REGION Network 20: Check connect giữa PLC với Server và HMI
   RUNG wire#powerrail
      Contact( "AlwaysTRUE" )
      "CheckConnectPLCServer_DB"(Signal := wire#w1, "Timeout(s)" := 60, Status => "DB_DataHMI".StatusConnectServer)
   END_RUNG
   RUNG wire#powerrail
      Contact( "AlwaysTRUE" )
      Contact( "DB_Server".ConnectPLC )
   END_RUNG wire#w1
   RUNG wire#powerrail
      Contact( "AlwaysTRUE" )
      Contact( "DB_Server".ConnectPLC )
      R_Coil( "DB_Server".ConnectPLC )
   END_RUNG
   RUNG wire#powerrail
      Contact( "AlwaysTRUE" )
      wire#w2
      "CreatePulse_DB_CheckConnectHMI"("pulse_on(x1ms)" := 1000, "pulse_off(x1ms)" := 1000, pulse => #pulse_check_connect_hmi)
   END_RUNG
   RUNG wire#w2
      P_Contact(operand := #pulse_check_connect_hmi, bit := "PulseP_Check_ConnectHmi")
      S_Coil( "DB_DataHMI".StatusConnectController )
   END_RUNG
   // the same network as SCL:
   IF "AlwaysTRUE" THEN
       "CheckConnectPLCServer_DB"(Signal := "AlwaysTRUE" AND "DB_Server".ConnectPLC,   // "CheckConnectPLCServer"
                               "Timeout(s)" := 60,
                               Status => "DB_DataHMI".StatusConnectServer);
   END_IF;
   IF "AlwaysTRUE" AND "DB_Server".ConnectPLC THEN "DB_Server".ConnectPLC := FALSE; END_IF;
   #_w1 := "AlwaysTRUE";
   IF #_w1 THEN
       "CreatePulse_DB_CheckConnectHMI"("pulse_on(x1ms)" := 1000,   // "CreatePulse"
                               "pulse_off(x1ms)" := 1000,
                               pulse => #pulse_check_connect_hmi);
   END_IF;
   #_w2 := #_w1 AND #pulse_check_connect_hmi AND NOT "PulseP_Check_ConnectHmi";   // rising edge of #pulse_check_connect_hmi
   "PulseP_Check_ConnectHmi" := #pulse_check_connect_hmi;
   IF #_w2 THEN "DB_DataHMI".StatusConnectController := TRUE; END_IF;
END_REGION

REGION Network 21: Reset Counter khi qua ca
   RUNG wire#powerrail
      Contact( "AlwaysTRUE" )
      Contact( "DB_Server".EventResetCounterInShift )
      wire#w1
      Add(in1 := "TagTest".NumberServerResetCounter, in2 := 1, out => "TagTest".NumberServerResetCounter)
      Move(in := 0, out1 => "DB_Machine".CounterMachineInShift)
      "ClearBufferLossInShift"()
   END_RUNG
   RUNG wire#w1
      R_Coil( "DB_Server".EventResetCounterInShift )
   END_RUNG
   // the same network as SCL:
   IF "AlwaysTRUE" AND "DB_Server".EventResetCounterInShift THEN
       "TagTest".NumberServerResetCounter := "TagTest".NumberServerResetCounter + 1;
       "DB_Machine".CounterMachineInShift := 0;
   END_IF;
   #_w1 := "AlwaysTRUE" AND "DB_Server".EventResetCounterInShift;
   IF #_w1 THEN
       "ClearBufferLossInShift"();
       "DB_Server".EventResetCounterInShift := FALSE;
   END_IF;
END_REGION

REGION Network 22: //////////////////End//////////////////
END_REGION

REGION Network 23: Test tính Speed
END_REGION

REGION Network 24 (SCL): Random Buffer Test
   IF "TagTest".TestRandomSparePart THEN
       "DB_Server".PageDataSparePart.MaxPage := 10;
       "DB_Server".ActionSearchLossSparePart := 2;
       "DB_Server".PageDataSparePart.TotalData := "DB_Server".PageDataSparePart.MaxPage * 30;

       FOR #index_for := 1 TO 30 DO
           #id_test := ("DB_Server".PageDataSparePart.PageCurrent - 1) * 30 + #index_for;

           "BufferServerSend".buffer_spare_part[#index_for].name := CONCAT(IN1 := 'Thiet bi: ', IN2 := UDINT_TO_STRING(#id_test));
           "BufferServerSend".buffer_spare_part[#index_for].start_time := "GlobalDB_RTC".RTC_Local;
           "BufferServerSend".buffer_spare_part[#index_for].end_time := "GlobalDB_RTC".RTC_Local;
           "BufferServerSend".buffer_spare_part[#index_for].product_count := #id_test;
       END_FOR;
   END_IF;


   IF "TagTest".TestRandomHistorical THEN
       FOR #index_for := 1 TO 50 DO
           #id_test := ("DB_Server".PageHistorical.PageCurrent - 1) * 50 + #index_for;

           "BuffersLoss_DB".buffer_loss_in_historical[#index_for].id := #id_test;
           "BuffersLoss_DB".buffer_loss_in_historical[#index_for].duration := #id_test * 10;
           "BuffersLoss_DB".buffer_loss_in_historical[#index_for].startTime := "GlobalDB_RTC".RTC_Local;
           "BuffersLoss_DB".buffer_loss_in_historical[#index_for].endTime := "GlobalDB_RTC".RTC_Local;
           "BuffersLoss_DB".buffer_loss_in_historical[#index_for].losscode := 0;
           "BuffersLoss_DB".buffer_loss_in_historical[#index_for].statusServer := 0;
       END_FOR;
   END_IF;
END_REGION

REGION Network 25: Clear Buffer To Test
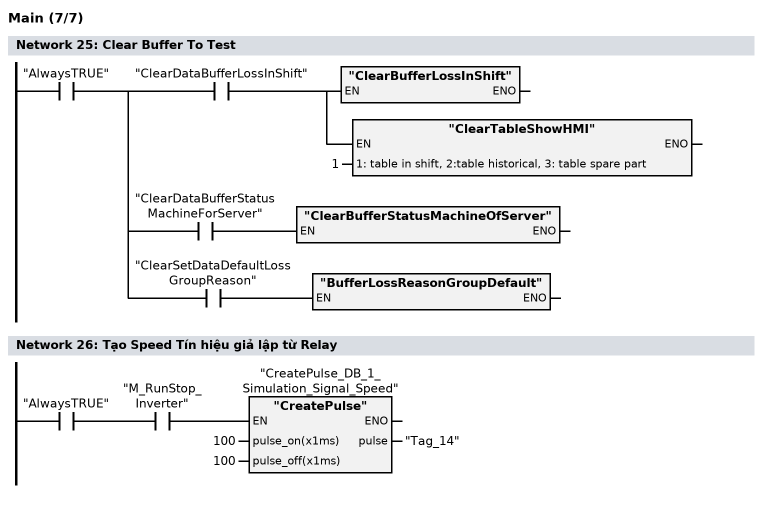
   RUNG wire#powerrail
      Contact( "AlwaysTRUE" )
      wire#w1
      Contact( "ClearDataBufferLossInShift" )
      wire#w2
      "ClearBufferLossInShift"()
   END_RUNG
   RUNG wire#w2
      "ClearTableShowHMI"("1: table in shift, 2:table historical, 3: table spare part" := 1)
   END_RUNG
   RUNG wire#w1
      Contact( "ClearDataBufferStatusMachineForServer" )
      "ClearBufferStatusMachineOfServer"()
   END_RUNG
   RUNG wire#w1
      Contact( "ClearSetDataDefaultLossGroupReason" )
      "BufferLossReasonGroupDefault"()
   END_RUNG
   // the same network as SCL:
   #_w1 := "AlwaysTRUE";
   #_w2 := "AlwaysTRUE" AND "ClearDataBufferLossInShift";
   IF #_w2 THEN
       "ClearBufferLossInShift"();
       "ClearTableShowHMI"("1: table in shift, 2:table historical, 3: table spare part" := 1);
   END_IF;
   IF #_w1 AND "ClearDataBufferStatusMachineForServer" THEN "ClearBufferStatusMachineOfServer"(); END_IF;
   IF #_w1 AND "ClearSetDataDefaultLossGroupReason" THEN "BufferLossReasonGroupDefault"(); END_IF;
END_REGION

REGION Network 26: Tạo Speed Tín hiệu giả lập từ Relay
   RUNG wire#powerrail
      Contact( "AlwaysTRUE" )
      Contact( "M_RunStop_Inverter" )
      "CreatePulse_DB_1_Simulation_Signal_Speed"("pulse_on(x1ms)" := 100, "pulse_off(x1ms)" := 100, pulse => "Tag_14")
   END_RUNG
   // the same network as SCL:
   IF "AlwaysTRUE" AND "M_RunStop_Inverter" THEN
       "CreatePulse_DB_1_Simulation_Signal_Speed"("pulse_on(x1ms)" := 100,   // "CreatePulse"
                               "pulse_off(x1ms)" := 100,
                               pulse => "Tag_14");
   END_IF;
END_REGION
END_ORGANIZATION_BLOCK

ORGANIZATION_BLOCK "InterrupTimer10ms(Simulation)"   // OB30, LAD, CyclicInterrupt
{ S7_Optimized_Access := 'TRUE' }
VERSION : 0.1
   VAR_INPUT
      Initial_Call : Bool;   // Initial call of this OB
      Event_Count : Int;   // Events discarded
   END_VAR
BEGIN

REGION Network 1: Tạo xung simulation cho sensors
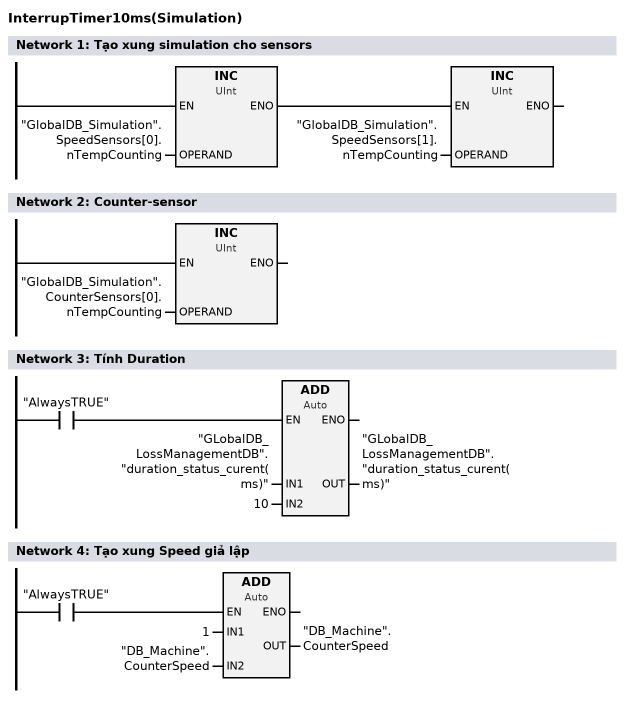
   RUNG wire#powerrail
      { S7_Templates := "DestType := UInt" } Inc( "GlobalDB_Simulation".SpeedSensors[0].nTempCounting )
      { S7_Templates := "DestType := UInt" } Inc( "GlobalDB_Simulation".SpeedSensors[1].nTempCounting )
   END_RUNG
   // the same network as SCL:
   "GlobalDB_Simulation".SpeedSensors[0].nTempCounting := "GlobalDB_Simulation".SpeedSensors[0].nTempCounting + 1;
   "GlobalDB_Simulation".SpeedSensors[1].nTempCounting := "GlobalDB_Simulation".SpeedSensors[1].nTempCounting + 1;
END_REGION

REGION Network 2: Counter-sensor
   RUNG wire#powerrail
      { S7_Templates := "DestType := UInt" } Inc( "GlobalDB_Simulation".CounterSensors[0].nTempCounting )
   END_RUNG
   // the same network as SCL:
   "GlobalDB_Simulation".CounterSensors[0].nTempCounting := "GlobalDB_Simulation".CounterSensors[0].nTempCounting + 1;
END_REGION

REGION Network 3: Tính Duration
   RUNG wire#powerrail
      Contact( "AlwaysTRUE" )
      Add(in1 := "GLobalDB_LossManagementDB"."duration_status_curent(ms)", in2 := 10, out => "GLobalDB_LossManagementDB"."duration_status_curent(ms)")
   END_RUNG
   // the same network as SCL:
   IF "AlwaysTRUE" THEN
       "GLobalDB_LossManagementDB"."duration_status_curent(ms)" := "GLobalDB_LossManagementDB"."duration_status_curent(ms)" + 10;
   END_IF;
END_REGION

REGION Network 4: Tạo xung Speed giả lập
   RUNG wire#powerrail
      Contact( "AlwaysTRUE" )
      Add(in1 := 1, in2 := "DB_Machine".CounterSpeed, out => "DB_Machine".CounterSpeed)
   END_RUNG
   // the same network as SCL:
   IF "AlwaysTRUE" THEN "DB_Machine".CounterSpeed := 1 + "DB_Machine".CounterSpeed; END_IF;
END_REGION
END_ORGANIZATION_BLOCK

ORGANIZATION_BLOCK "Interrupt Analog Cyclic"   // OB31, LAD, CyclicInterrupt
{ S7_Optimized_Access := 'TRUE' }
VERSION : 0.1
   VAR_INPUT
      Initial_Call : Bool;   // Initial call of this OB
      Event_Count : Int;   // Events discarded
   END_VAR
   VAR CONSTANT
      MAX_IDX : Int := 3;
   END_VAR
   VAR_TEMP   // added for the SCL form of the ladder/FBD networks
      _w1 : Bool;
      _w2 : Bool;
   END_VAR
BEGIN

REGION Network 1: Check Index
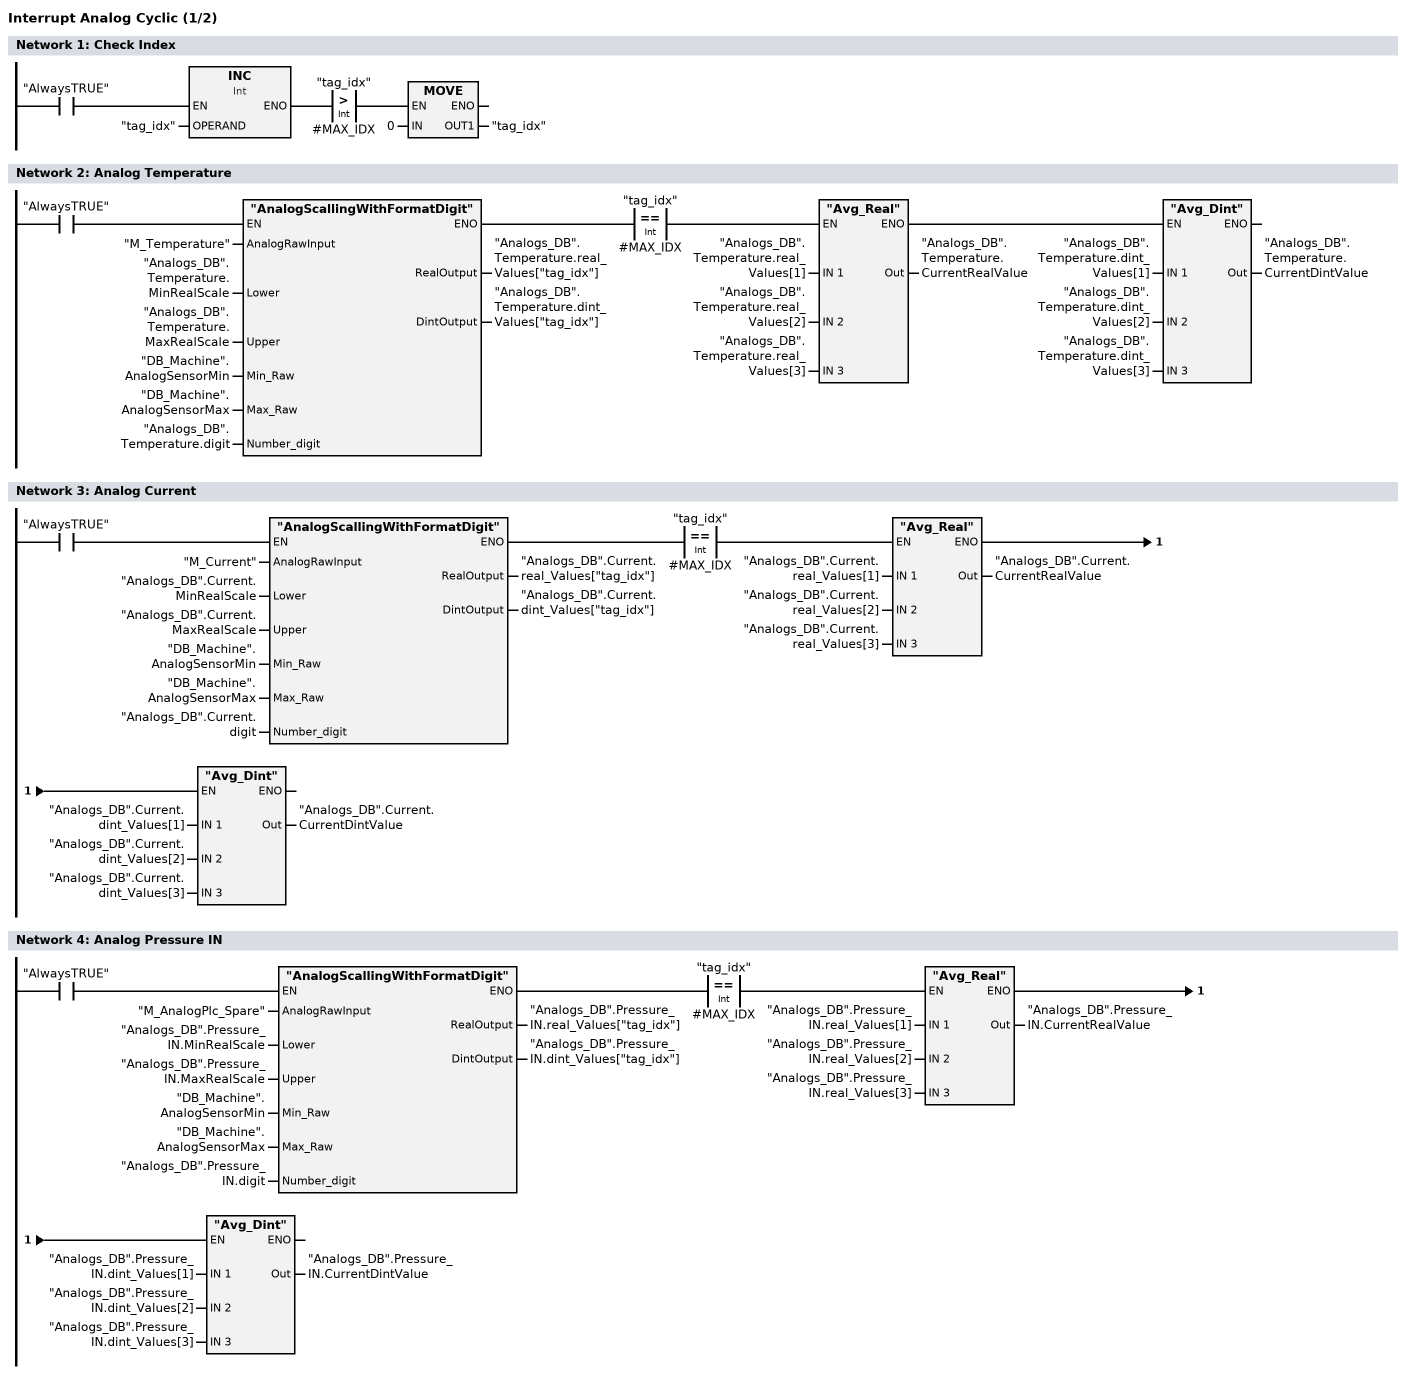
   RUNG wire#powerrail
      Contact( "AlwaysTRUE" )
      { S7_Templates := "DestType := Int" } Inc( "tag_idx" )
      { S7_Templates := "SrcType := Int" } GT_Contact(in1 := "tag_idx", in2 := #MAX_IDX)
      Move(in := 0, out1 => "tag_idx")
   END_RUNG
   // the same network as SCL:
   IF "AlwaysTRUE" THEN "tag_idx" := "tag_idx" + 1; END_IF;
   IF "AlwaysTRUE" AND ("tag_idx" > #MAX_IDX) THEN "tag_idx" := 0; END_IF;
END_REGION

REGION Network 2: Analog Temperature
   RUNG wire#powerrail
      Contact( "AlwaysTRUE" )
      "AnalogScallingWithFormatDigit"(AnalogRawInput := "M_Temperature", Lower := "Analogs_DB".Temperature.MinRealScale, Upper := "Analogs_DB".Temperature.MaxRealScale, Min_Raw := "DB_Machine".AnalogSensorMin, Max_Raw := "DB_Machine".AnalogSensorMax, Number_digit := "Analogs_DB".Temperature.digit, RealOutput => "Analogs_DB".Temperature.real_Values["tag_idx"], DintOutput => "Analogs_DB".Temperature.dint_Values["tag_idx"])
      { S7_Templates := "SrcType := Int" } EQ_Contact(in1 := "tag_idx", in2 := #MAX_IDX)
      "Avg_Real"("IN 1" := "Analogs_DB".Temperature.real_Values[1], "IN 2" := "Analogs_DB".Temperature.real_Values[2], "IN 3" := "Analogs_DB".Temperature.real_Values[3], Out => "Analogs_DB".Temperature.CurrentRealValue)
      "Avg_Dint"("IN 1" := "Analogs_DB".Temperature.dint_Values[1], "IN 2" := "Analogs_DB".Temperature.dint_Values[2], "IN 3" := "Analogs_DB".Temperature.dint_Values[3], Out => "Analogs_DB".Temperature.CurrentDintValue)
   END_RUNG
   // the same network as SCL:
   "AnalogScallingWithFormatDigit"(EN := "AlwaysTRUE",
                           AnalogRawInput := "M_Temperature",
                           Lower := "Analogs_DB".Temperature.MinRealScale,
                           Upper := "Analogs_DB".Temperature.MaxRealScale,
                           Min_Raw := "DB_Machine".AnalogSensorMin,
                           Max_Raw := "DB_Machine".AnalogSensorMax,
                           Number_digit := "Analogs_DB".Temperature.digit,
                           RealOutput => "Analogs_DB".Temperature.real_Values["tag_idx"],
                           DintOutput => "Analogs_DB".Temperature.dint_Values["tag_idx"],
                           ENO => #_w1);
   "Avg_Real"(EN := #_w1 AND ("tag_idx" = #MAX_IDX),
              "IN 1" := "Analogs_DB".Temperature.real_Values[1],
              "IN 2" := "Analogs_DB".Temperature.real_Values[2],
              "IN 3" := "Analogs_DB".Temperature.real_Values[3],
              Out => "Analogs_DB".Temperature.CurrentRealValue,
              ENO => #_w2);
   IF #_w2 THEN
       "Avg_Dint"("IN 1" := "Analogs_DB".Temperature.dint_Values[1],
                  "IN 2" := "Analogs_DB".Temperature.dint_Values[2],
                  "IN 3" := "Analogs_DB".Temperature.dint_Values[3],
                  Out => "Analogs_DB".Temperature.CurrentDintValue);
   END_IF;
END_REGION

REGION Network 3: Analog Current
   RUNG wire#powerrail
      Contact( "AlwaysTRUE" )
      "AnalogScallingWithFormatDigit"(AnalogRawInput := "M_Current", Lower := "Analogs_DB".Current.MinRealScale, Upper := "Analogs_DB".Current.MaxRealScale, Min_Raw := "DB_Machine".AnalogSensorMin, Max_Raw := "DB_Machine".AnalogSensorMax, Number_digit := "Analogs_DB".Current.digit, RealOutput => "Analogs_DB".Current.real_Values["tag_idx"], DintOutput => "Analogs_DB".Current.dint_Values["tag_idx"])
      { S7_Templates := "SrcType := Int" } EQ_Contact(in1 := "tag_idx", in2 := #MAX_IDX)
      "Avg_Real"("IN 1" := "Analogs_DB".Current.real_Values[1], "IN 2" := "Analogs_DB".Current.real_Values[2], "IN 3" := "Analogs_DB".Current.real_Values[3], Out => "Analogs_DB".Current.CurrentRealValue)
      "Avg_Dint"("IN 1" := "Analogs_DB".Current.dint_Values[1], "IN 2" := "Analogs_DB".Current.dint_Values[2], "IN 3" := "Analogs_DB".Current.dint_Values[3], Out => "Analogs_DB".Current.CurrentDintValue)
   END_RUNG
   // the same network as SCL:
   "AnalogScallingWithFormatDigit"(EN := "AlwaysTRUE",
                           AnalogRawInput := "M_Current",
                           Lower := "Analogs_DB".Current.MinRealScale,
                           Upper := "Analogs_DB".Current.MaxRealScale,
                           Min_Raw := "DB_Machine".AnalogSensorMin,
                           Max_Raw := "DB_Machine".AnalogSensorMax,
                           Number_digit := "Analogs_DB".Current.digit,
                           RealOutput => "Analogs_DB".Current.real_Values["tag_idx"],
                           DintOutput => "Analogs_DB".Current.dint_Values["tag_idx"],
                           ENO => #_w1);
   "Avg_Real"(EN := #_w1 AND ("tag_idx" = #MAX_IDX),
              "IN 1" := "Analogs_DB".Current.real_Values[1],
              "IN 2" := "Analogs_DB".Current.real_Values[2],
              "IN 3" := "Analogs_DB".Current.real_Values[3],
              Out => "Analogs_DB".Current.CurrentRealValue,
              ENO => #_w2);
   IF #_w2 THEN
       "Avg_Dint"("IN 1" := "Analogs_DB".Current.dint_Values[1],
                  "IN 2" := "Analogs_DB".Current.dint_Values[2],
                  "IN 3" := "Analogs_DB".Current.dint_Values[3],
                  Out => "Analogs_DB".Current.CurrentDintValue);
   END_IF;
END_REGION

REGION Network 4: Analog Pressure IN
   RUNG wire#powerrail
      Contact( "AlwaysTRUE" )
      "AnalogScallingWithFormatDigit"(AnalogRawInput := "M_AnalogPlc_Spare", Lower := "Analogs_DB".Pressure_IN.MinRealScale, Upper := "Analogs_DB".Pressure_IN.MaxRealScale, Min_Raw := "DB_Machine".AnalogSensorMin, Max_Raw := "DB_Machine".AnalogSensorMax, Number_digit := "Analogs_DB".Pressure_IN.digit, RealOutput => "Analogs_DB".Pressure_IN.real_Values["tag_idx"], DintOutput => "Analogs_DB".Pressure_IN.dint_Values["tag_idx"])
      { S7_Templates := "SrcType := Int" } EQ_Contact(in1 := "tag_idx", in2 := #MAX_IDX)
      "Avg_Real"("IN 1" := "Analogs_DB".Pressure_IN.real_Values[1], "IN 2" := "Analogs_DB".Pressure_IN.real_Values[2], "IN 3" := "Analogs_DB".Pressure_IN.real_Values[3], Out => "Analogs_DB".Pressure_IN.CurrentRealValue)
      "Avg_Dint"("IN 1" := "Analogs_DB".Pressure_IN.dint_Values[1], "IN 2" := "Analogs_DB".Pressure_IN.dint_Values[2], "IN 3" := "Analogs_DB".Pressure_IN.dint_Values[3], Out => "Analogs_DB".Pressure_IN.CurrentDintValue)
   END_RUNG
   // the same network as SCL:
   "AnalogScallingWithFormatDigit"(EN := "AlwaysTRUE",
                           AnalogRawInput := "M_AnalogPlc_Spare",
                           Lower := "Analogs_DB".Pressure_IN.MinRealScale,
                           Upper := "Analogs_DB".Pressure_IN.MaxRealScale,
                           Min_Raw := "DB_Machine".AnalogSensorMin,
                           Max_Raw := "DB_Machine".AnalogSensorMax,
                           Number_digit := "Analogs_DB".Pressure_IN.digit,
                           RealOutput => "Analogs_DB".Pressure_IN.real_Values["tag_idx"],
                           DintOutput => "Analogs_DB".Pressure_IN.dint_Values["tag_idx"],
                           ENO => #_w1);
   "Avg_Real"(EN := #_w1 AND ("tag_idx" = #MAX_IDX),
              "IN 1" := "Analogs_DB".Pressure_IN.real_Values[1],
              "IN 2" := "Analogs_DB".Pressure_IN.real_Values[2],
              "IN 3" := "Analogs_DB".Pressure_IN.real_Values[3],
              Out => "Analogs_DB".Pressure_IN.CurrentRealValue,
              ENO => #_w2);
   IF #_w2 THEN
       "Avg_Dint"("IN 1" := "Analogs_DB".Pressure_IN.dint_Values[1],
                  "IN 2" := "Analogs_DB".Pressure_IN.dint_Values[2],
                  "IN 3" := "Analogs_DB".Pressure_IN.dint_Values[3],
                  Out => "Analogs_DB".Pressure_IN.CurrentDintValue);
   END_IF;
END_REGION

REGION Network 5: Analog Pressure OUT
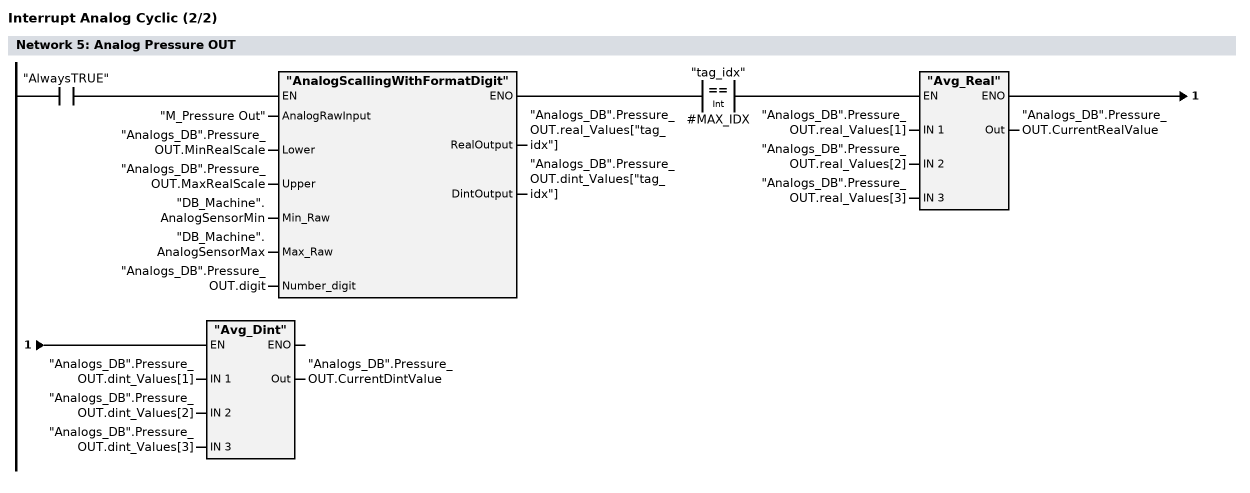
   RUNG wire#powerrail
      Contact( "AlwaysTRUE" )
      "AnalogScallingWithFormatDigit"(AnalogRawInput := "M_Pressure Out", Lower := "Analogs_DB".Pressure_OUT.MinRealScale, Upper := "Analogs_DB".Pressure_OUT.MaxRealScale, Min_Raw := "DB_Machine".AnalogSensorMin, Max_Raw := "DB_Machine".AnalogSensorMax, Number_digit := "Analogs_DB".Pressure_OUT.digit, RealOutput => "Analogs_DB".Pressure_OUT.real_Values["tag_idx"], DintOutput => "Analogs_DB".Pressure_OUT.dint_Values["tag_idx"])
      { S7_Templates := "SrcType := Int" } EQ_Contact(in1 := "tag_idx", in2 := #MAX_IDX)
      "Avg_Real"("IN 1" := "Analogs_DB".Pressure_OUT.real_Values[1], "IN 2" := "Analogs_DB".Pressure_OUT.real_Values[2], "IN 3" := "Analogs_DB".Pressure_OUT.real_Values[3], Out => "Analogs_DB".Pressure_OUT.CurrentRealValue)
      "Avg_Dint"("IN 1" := "Analogs_DB".Pressure_OUT.dint_Values[1], "IN 2" := "Analogs_DB".Pressure_OUT.dint_Values[2], "IN 3" := "Analogs_DB".Pressure_OUT.dint_Values[3], Out => "Analogs_DB".Pressure_OUT.CurrentDintValue)
   END_RUNG
   // the same network as SCL:
   "AnalogScallingWithFormatDigit"(EN := "AlwaysTRUE",
                           AnalogRawInput := "M_Pressure Out",
                           Lower := "Analogs_DB".Pressure_OUT.MinRealScale,
                           Upper := "Analogs_DB".Pressure_OUT.MaxRealScale,
                           Min_Raw := "DB_Machine".AnalogSensorMin,
                           Max_Raw := "DB_Machine".AnalogSensorMax,
                           Number_digit := "Analogs_DB".Pressure_OUT.digit,
                           RealOutput => "Analogs_DB".Pressure_OUT.real_Values["tag_idx"],
                           DintOutput => "Analogs_DB".Pressure_OUT.dint_Values["tag_idx"],
                           ENO => #_w1);
   "Avg_Real"(EN := #_w1 AND ("tag_idx" = #MAX_IDX),
              "IN 1" := "Analogs_DB".Pressure_OUT.real_Values[1],
              "IN 2" := "Analogs_DB".Pressure_OUT.real_Values[2],
              "IN 3" := "Analogs_DB".Pressure_OUT.real_Values[3],
              Out => "Analogs_DB".Pressure_OUT.CurrentRealValue,
              ENO => #_w2);
   IF #_w2 THEN
       "Avg_Dint"("IN 1" := "Analogs_DB".Pressure_OUT.dint_Values[1],
                  "IN 2" := "Analogs_DB".Pressure_OUT.dint_Values[2],
                  "IN 3" := "Analogs_DB".Pressure_OUT.dint_Values[3],
                  Out => "Analogs_DB".Pressure_OUT.CurrentDintValue);
   END_IF;
END_REGION
END_ORGANIZATION_BLOCK

ORGANIZATION_BLOCK "Speed_Cyclic_Interrupt_2s"   // OB32, LAD, CyclicInterrupt
{ S7_Optimized_Access := 'TRUE' }
VERSION : 0.1
   VAR_INPUT
      Initial_Call : Bool;   // Initial call of this OB
      Event_Count : Int;   // Events discarded
   END_VAR
   VAR_TEMP   // added for the SCL form of the ladder/FBD networks
      _w1 : Bool;
   END_VAR
BEGIN

REGION Network 1
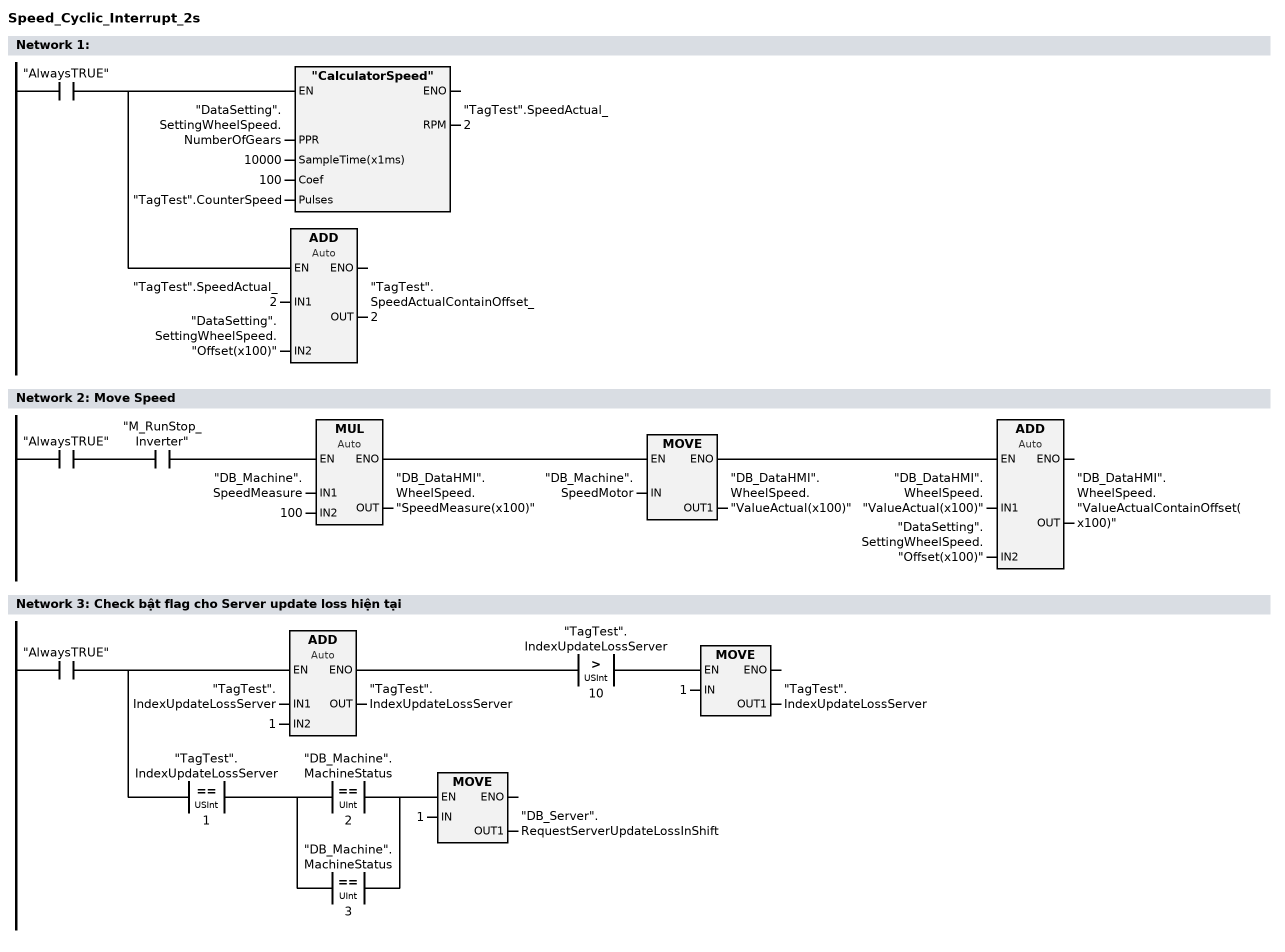
   RUNG wire#powerrail
      Contact( "AlwaysTRUE" )
      wire#w1
      "CalculatorSpeed"(PPR := "DataSetting".SettingWheelSpeed.NumberOfGears, "SampleTime(x1ms)" := 10000, Coef := 100, Pulses := "TagTest".CounterSpeed, RPM => "TagTest".SpeedActual_2)
   END_RUNG
   RUNG wire#w1
      Add(in1 := "TagTest".SpeedActual_2, in2 := "DataSetting".SettingWheelSpeed."Offset(x100)", out => "TagTest".SpeedActualContainOffset_2)
   END_RUNG
   // the same network as SCL:
   #_w1 := "AlwaysTRUE";
   IF #_w1 THEN
       "CalculatorSpeed"(PPR := "DataSetting".SettingWheelSpeed.NumberOfGears,
                         "SampleTime(x1ms)" := 10000,
                         Coef := 100,
                         Pulses := "TagTest".CounterSpeed,
                         RPM => "TagTest".SpeedActual_2);
       "TagTest".SpeedActualContainOffset_2 := "TagTest".SpeedActual_2 + "DataSetting".SettingWheelSpeed."Offset(x100)";
   END_IF;
END_REGION

REGION Network 2: Move Speed
   RUNG wire#powerrail
      Contact( "AlwaysTRUE" )
      Contact( "M_RunStop_Inverter" )
      Mul(in1 := "DB_Machine".SpeedMeasure, in2 := 100, out => "DB_DataHMI".WheelSpeed."SpeedMeasure(x100)")
      Move(in := "DB_Machine".SpeedMotor, out1 => "DB_DataHMI".WheelSpeed."ValueActual(x100)")
      Add(in1 := "DB_DataHMI".WheelSpeed."ValueActual(x100)", in2 := "DataSetting".SettingWheelSpeed."Offset(x100)", out => "DB_DataHMI".WheelSpeed."ValueActualContainOffset(x100)")
   END_RUNG
   // the same network as SCL:
   IF "AlwaysTRUE" AND "M_RunStop_Inverter" THEN
       "DB_DataHMI".WheelSpeed."SpeedMeasure(x100)" := "DB_Machine".SpeedMeasure * 100;
       "DB_DataHMI".WheelSpeed."ValueActual(x100)" := "DB_Machine".SpeedMotor;
       "DB_DataHMI".WheelSpeed."ValueActualContainOffset(x100)" := "DB_DataHMI".WheelSpeed."ValueActual(x100)" + "DataSetting".SettingWheelSpeed."Offset(x100)";
   END_IF;
END_REGION

REGION Network 3: Check bật flag cho Server update loss hiện tại
   RUNG wire#powerrail
      Contact( "AlwaysTRUE" )
      wire#w1
      Add(in1 := "TagTest".IndexUpdateLossServer, in2 := 1, out => "TagTest".IndexUpdateLossServer)
      { S7_Templates := "SrcType := USInt" } GT_Contact(in1 := "TagTest".IndexUpdateLossServer, in2 := 10)
      Move(in := 1, out1 => "TagTest".IndexUpdateLossServer)
   END_RUNG
   RUNG wire#w1
      { S7_Templates := "SrcType := USInt" } EQ_Contact(in1 := "TagTest".IndexUpdateLossServer, in2 := 1)
      wire#w2
      { S7_Templates := "SrcType := UInt" } EQ_Contact(in1 := "DB_Machine".MachineStatus, in2 := 2)
      wire#w3
      Move(in := 1, out1 => "DB_Server".RequestServerUpdateLossInShift)
   END_RUNG
   RUNG wire#w2
      { S7_Templates := "SrcType := UInt" } EQ_Contact(in1 := "DB_Machine".MachineStatus, in2 := 3)
   END_RUNG wire#w3
   // the same network as SCL:
   IF "AlwaysTRUE" THEN "TagTest".IndexUpdateLossServer := "TagTest".IndexUpdateLossServer + 1; END_IF;
   IF "AlwaysTRUE" AND ("TagTest".IndexUpdateLossServer > 10) THEN
       "TagTest".IndexUpdateLossServer := 1;
   END_IF;
   IF "AlwaysTRUE" AND ("TagTest".IndexUpdateLossServer = 1) AND (("DB_Machine".MachineStatus = 2) OR ("DB_Machine".MachineStatus = 3)) THEN
       "DB_Server".RequestServerUpdateLossInShift := 1;
   END_IF;
END_REGION
END_ORGANIZATION_BLOCK

ORGANIZATION_BLOCK "RandomSensor"   // OB33, LAD, CyclicInterrupt
{ S7_Optimized_Access := 'TRUE' }
VERSION : 0.1
   VAR_INPUT
      Initial_Call : Bool;   // Initial call of this OB
      Event_Count : Int;   // Events discarded
   END_VAR
   VAR_TEMP
      pulse_random_speed : Bool;
   END_VAR
BEGIN

REGION Network 1 (SCL): Random Analog
   // IF "TagTest".RandomAnalog THEN
   //     "RandomAnalogs".IndexRandom += 1;
   //     "RandomAnalogs".ValueTemp := "RandomAnalogs".ValueTemp * 214013 + 2531011;

   //     //Current
   //     "RandomAnalogs".from_random := 16500;
   //     "RandomAnalogs".to_random := 17000;
   //     "RandomAnalogs".Current_Analog := ABS("RandomAnalogs".ValueTemp MOD ( "RandomAnalogs".to_random - "RandomAnalogs".from_random + 1)) + "RandomAnalogs".from_random;

   //     //Temp
   //     "RandomAnalogs".from_random := 15500;
   //     "RandomAnalogs".to_random := 16500;
   //     "RandomAnalogs".Temp_Analog := ABS("RandomAnalogs".ValueTemp MOD ("RandomAnalogs".to_random - "RandomAnalogs".from_random + 1)) + "RandomAnalogs".from_random;

   //     //Pressure
   //     "RandomAnalogs".from_random := 14000;
   //     "RandomAnalogs".to_random := 14100;
   //     "RandomAnalogs".Pressure_Analog := ABS("RandomAnalogs".ValueTemp MOD ("RandomAnalogs".to_random - "RandomAnalogs".from_random + 1)) + "RandomAnalogs".from_random;

   //     //Speed
   //     "RandomAnalogs".from_random := 1700;
   //     "RandomAnalogs".to_random := 1705;
   //     "RandomAnalogs".Speed_Value := ABS("RandomAnalogs".ValueTemp MOD ("RandomAnalogs".to_random - "RandomAnalogs".from_random + 1)) + "RandomAnalogs".from_random;

   //     // IF "RandomAnalogs".IndexRandom = 1 THEN
   //     //     "RandomAnalogs".Speed_Value := ABS("RandomAnalogs".Speed_Value MOD 51);
   //     // // ELSIF "RandomAnalogs".IndexRandom = 2 THEN
   //     // //     "RandomAnalogs".Current_Analog := ABS("RandomAnalogs".ValueTemp MOD ("DB_Machine".AnalogSensorMax - "DB_Machine".AnalogSensorMin + 1)) + "DB_Machine".AnalogSensorMin;
   //     // ELSIF "RandomAnalogs".IndexRandom = 3 THEN
   //     //     "RandomAnalogs".Temp_Analog := ABS("RandomAnalogs".ValueTemp MOD ("DB_Machine".AnalogSensorMax - "DB_Machine".AnalogSensorMin + 1)) + "DB_Machine".AnalogSensorMin;
   //     // ELSIF "RandomAnalogs".IndexRandom = 4 THEN
   //     //     "RandomAnalogs".Pressure_Analog := ABS("RandomAnalogs".ValueTemp MOD ("DB_Machine".AnalogSensorMax - "DB_Machine".AnalogSensorMin + 1)) + "DB_Machine".AnalogSensorMin;
   //     // ELSIF "RandomAnalogs".IndexRandom > 4 OR "RandomAnalogs".IndexRandom < 1 THEN
   //     //     "RandomAnalogs".IndexRandom := 0;
   //     // END_IF;
   // END_IF;
END_REGION
END_ORGANIZATION_BLOCK

ORGANIZATION_BLOCK "Interrupt Speed Sensor P"   // OB40, LAD, HWProcessInterrupt
{ S7_Optimized_Access := 'TRUE' }
VERSION : 0.1
   VAR_INPUT
      LADDR : Hw_Io;   // Hardware identifier
      USI : Word;   // User structure identifier
      IChannel : USInt;   // Interrupt channel number
      EventType : Byte;   // EventType
   END_VAR
BEGIN

REGION Network 1: Cách 1
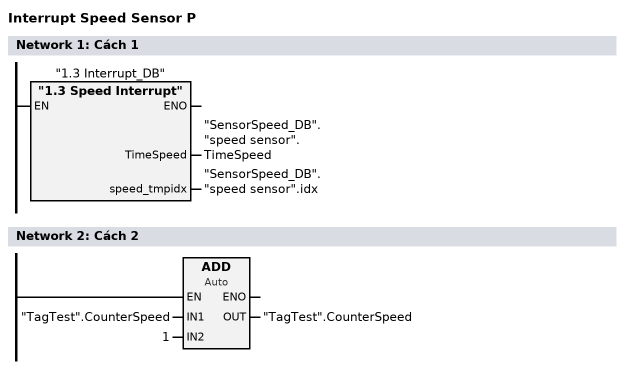
   RUNG wire#powerrail
      "1.3 Interrupt_DB"(TimeSpeed => "SensorSpeed_DB"."speed sensor".TimeSpeed, speed_tmpidx => "SensorSpeed_DB"."speed sensor".idx)
   END_RUNG
   // the same network as SCL:
   "1.3 Interrupt_DB"(TimeSpeed => "SensorSpeed_DB"."speed sensor".TimeSpeed,   // "1.3 Speed Interrupt"
                      speed_tmpidx => "SensorSpeed_DB"."speed sensor".idx);
END_REGION

REGION Network 2: Cách 2
   RUNG wire#powerrail
      Add(in1 := "TagTest".CounterSpeed, in2 := 1, out => "TagTest".CounterSpeed)
   END_RUNG
   // the same network as SCL:
   "TagTest".CounterSpeed := "TagTest".CounterSpeed + 1;
END_REGION
END_ORGANIZATION_BLOCK

ORGANIZATION_BLOCK "Startup"   // OB100, SCL, Startup
TITLE = "Complete Restart"
{ S7_Optimized_Access := 'TRUE' }
VERSION : 0.1
   VAR_INPUT
      LostRetentive : Bool;   // True if retentive data are lost
      LostRTC : Bool;   // True if date and time are lost
   END_VAR
BEGIN
   /////////////////////////////////////////Load Setting Sensor Analog//////////////////////////////////////////////
   //Check tgian Show event, mặc định 5s
   IF "DataSetting"."TimeThresholdShowWarningAssignLoss(s)" = 0 THEN
       "DataSetting"."TimeThresholdShowWarningAssignLoss(s)" := 5;
   END_IF;

   /////////////////////////////////////////Load Setting Sensor vào DB Analog////////////////////////////////////////
   "MoveDataSettingToBufferAnalog"();

   /////////////////////////////////////////Load Setting Sensor vào DB HMI//////////////////////////////////////////
   "MoveDataSettingToHmi"();

   /////////////////////////////////////////Load Setting Sensor vào DB Server///////////////////////////////////////
   "MoveDataSettingToServer"();

   /////////////////////////////////////////////////Layer Type Previuous ///////////////////////////////////////////
   "DB_DataHMI".TypeLayer := "DataSetting".TypeLayer;

   //////////////////////////////Yêu cầu Server gửi thông tin Group và Description Loss/////////////////////////////
   "DB_Server".RequestServerWriteLossGroup_Reason := 1;

   ///////////////////////////Thông tin máy ///////////////////////
   "DataSetting".InforStation.Factory := 'Factory 1';
   "DataSetting".InforStation.Workshop := 'Workshop 1';
   "DataSetting".InforStation.LineName := 'Line 1';
   "DataSetting".InforStation.MachineName := 'Machine 1';
   // //"DataSetting".InforStation.MachineCode := 'machine1';

   // "DataSetting".InforStation.Factory := 'Factory 2';
   // "DataSetting".InforStation.Workshop := 'Workshop 2';
   // "DataSetting".InforStation.LineName := 'Line 2';
   // "DataSetting".InforStation.MachineName := 'Machine 2';
   // "DataSetting".InforStation.MachineCode := 'machine2';
   // 


   "TagTest".NumberOnPowerPLC += 1;
   "TagTest".TimeLastOnPlc := "TagTest".TimeLastOnPlcRealTime;
   //Xử lý case khi on điện lại PLC : Log lại status
   IF "StatusMachineSendServerDB".index_current >= "StatusMachineSendServerDB".min_index_buffer AND
       "StatusMachineSendServerDB".index_current <= "StatusMachineSendServerDB".max_index_buffer THEN //Kiểm tra Index nằm trong range buffer (1->100)
       //Thêm Status
       "StatusMachineSendServerDB".StatusMachineBuffer["StatusMachineSendServerDB".index_current].status := 4;
       "StatusMachineSendServerDB".StatusMachineBuffer["StatusMachineSendServerDB".index_current].time_start := "TagTest".TimeLastOnPlc;
       "StatusMachineSendServerDB".StatusMachineBuffer["StatusMachineSendServerDB".index_current].timer_end := "GlobalDB_RTC".RTC_Local;

       //Cập nhật Status cũ 
       IF "StatusMachineSendServerDB".index_current = "StatusMachineSendServerDB".min_index_buffer THEN
           "StatusMachineSendServerDB".StatusMachineBuffer["StatusMachineSendServerDB".max_index_buffer].timer_end :=  "TagTest".TimeLastOnPlc;
       ELSE
           "StatusMachineSendServerDB".StatusMachineBuffer["StatusMachineSendServerDB".index_current - 1].timer_end :=  "TagTest".TimeLastOnPlc;
       END_IF;

       //Tăng Index buffer
       "StatusMachineSendServerDB".index_current += 1;
       IF "StatusMachineSendServerDB".index_current > "StatusMachineSendServerDB".max_index_buffer THEN
           "StatusMachineSendServerDB".index_current := 1;
       END_IF;

       //On flag bit Server để check đồng bộ lại data
       "DB_Server".RequestServerUpdateBufferStatusMachine := 1;
   ELSE //nếu nằm ngoài range buffer thì mặc định bằng 1
       "StatusMachineSendServerDB".index_current := 1;
   END_IF;

   //"GLobalDB_LossManagementDB"."duration_status_curent(ms)" := 0;
END_ORGANIZATION_BLOCK

// folder: Analogs

FUNCTION "CheckAlarmSensor" : Void   // FC19, SCL
{ S7_Optimized_Access := 'TRUE' }
VERSION : 0.1
   VAR_INPUT
      Value : DInt;
      LowerSetting : DInt;
      UpperSetting : DInt;
   END_VAR
   VAR_OUTPUT
      Alarm : UInt;   // 1: Oke; 2: > Upper; 3< Lower, NG
   END_VAR
BEGIN
   IF #Value < #LowerSetting THEN
       #Alarm := 3;
   ELSIF #Value > #UpperSetting THEN
       #Alarm := 2;
   ELSIF #Value <= #UpperSetting AND #Value >= #LowerSetting THEN
       #Alarm := 1;
   ELSE
       #Alarm := 0;
   END_IF;
END_FUNCTION

FUNCTION "CalculatorValueNotOffset" : Void   // FC52, SCL
{ S7_Optimized_Access := 'TRUE' }
VERSION : 0.1
   VAR_INPUT
      AnalogCurrent : DInt;
      AnalogMin : DInt;
      AnalogMax : DInt;
      "RangeSensorMin(x100)" : DInt;
      "RangeSensorMax(x100)" : DInt;
   END_VAR
   VAR_OUTPUT
      "Value(x100)" : DInt;
   END_VAR
   VAR_TEMP
      OffsetAnalog : DInt;
      OffsetSensor : DInt;
      Numerator : DInt;
   END_VAR
BEGIN
   IF #AnalogMin<=#AnalogMax AND
       #AnalogCurrent>= #AnalogMin AND #AnalogCurrent<=#AnalogMax AND
       #"RangeSensorMax(x100)">= #"RangeSensorMin(x100)" THEN

       #OffsetAnalog := #AnalogMax - #AnalogMin;
       #OffsetSensor := #"RangeSensorMax(x100)" - #"RangeSensorMin(x100)";
       #Numerator := #AnalogCurrent - #AnalogMin;

       IF #OffsetAnalog<>0 THEN
           #"Value(x100)" := (#Numerator * #OffsetSensor) / #OffsetAnalog + #"RangeSensorMin(x100)";
       ELSE
           #"Value(x100)" := #"RangeSensorMin(x100)";
       END_IF;
   ELSE
       #"Value(x100)" := 0;
   END_IF;
END_FUNCTION

FUNCTION "CvtUnitPressure" : Void   // FC59, SCL
{ S7_Optimized_Access := 'TRUE' }
VERSION : 0.1
   VAR_INPUT
      pressure_in : DInt;
      coef_unit : DInt;
   END_VAR
   VAR_OUTPUT
      pressure_out : DInt;
   END_VAR
BEGIN
   #pressure_out := REAL_TO_DINT(DINT_TO_REAL(#pressure_in) * DINT_TO_REAL(#coef_unit));
END_FUNCTION

// folder: Assignloss

FUNCTION "AssignLoss" : Void   // FC39, SCL
{ S7_Optimized_Access := 'TRUE' }
VERSION : 0.1
   VAR_INPUT
      index_row_assign : UInt;   // from 1 to 5
      "1: loss in shift - 2 loss historical" : USInt;   // 1: loss in shift - 2: loss historical
      index_select : UInt;   // from 1 to 10
   END_VAR
   VAR_TEMP
      id_assign : UDInt;
      index_for : USInt;
      loss_code_assign : UInt;
   END_VAR
BEGIN
   IF #index_row_assign>=1 AND #index_row_assign<=5 THEN
       IF #"1: loss in shift - 2 loss historical" = 1 THEN
           #id_assign := "DB_DataHMI".DataLossInShiftShowHmiDTO[#index_row_assign].id;

           #loss_code_assign := "DB_DataHMI".LossDescriptionHmiDTO[#index_select].index_buffer;

           FOR #index_for := 1 TO 100 DO
               IF "BuffersLoss_DB".buffer_loss_in_shift[#index_for].id = #id_assign THEN
                   "BuffersLoss_DB".buffer_loss_in_shift[#index_for].losscode := #loss_code_assign;
                   //"BuffersLoss_DB".buffer_loss_in_shift[#index_for].statusServer := 1;

                   //Yêu cầu Server Update
                   "DB_Server".RequestServerUpdateLossInShift := 1;
                   EXIT;
               END_IF;
           END_FOR;
       ELSIF #"1: loss in shift - 2 loss historical" = 2 THEN
           #loss_code_assign := "DB_DataHMI".LossDescriptionHmiDTO[#index_select].index_buffer;

           #id_assign := #index_row_assign + ("DB_DataHMI".PageDataLossHistorical.PageCurrent - ("DB_Server".PageHistorical.PageCurrent-1)*10-1) * 5;
           "BuffersLoss_DB".buffer_loss_in_historical[#id_assign].losscode := #loss_code_assign;

           //Yêu cầu Server Update
           "DB_Server".RequestServerUpdateLossHistorical := 1;

           // #id_assign := "DB_DataHMI".DataLossHistoricalShowHmiDTO[#index_row_assign].id;
           // FOR #index_for := 1 TO 50 DO
           //     IF "BuffersLoss_DB".buffer_loss_in_historical[#index_for].id = #id_assign THEN
           //         "BuffersLoss_DB".buffer_loss_in_historical[#index_for].losscode := #loss_code_assign;
           //         //"BuffersLoss_DB".buffer_loss_in_historical[#index_for].statusServer := 1;

           //         //Yêu cầu Server Update
           //         "DB_Server".RequestServerUpdateLossHistorical := 1;
           //         EXIT;
           //     END_IF;
           // END_FOR;
       END_IF;
   END_IF;

   "DB_DataHMI".LossGroupSelectId := 0;
   "DB_DataHMI".LossReasonSelectId := 0;
END_FUNCTION

FUNCTION "CheckShowDataHistorical" : Void   // FC54, SCL
{ S7_Optimized_Access := 'TRUE' }
VERSION : 0.1
   VAR_INPUT
      PageMaxHMI : UDInt;
      PageCurrentHMI : UDInt;
      PageCurrentRequestServer : UDInt;
   END_VAR
   VAR_TEMP
      index_buffer : UDInt;
      index_for : USInt;
      page_current_server : UDInt;
   END_VAR
BEGIN
   //Move ngày Serach
   "DB_Server".SearchDataLossHistorical := "DB_DataHMI".SearchDataLoss;

   IF #PageCurrentHMI >= 1 AND #PageCurrentRequestServer >= 1 AND #PageMaxHMI >= 1 THEN
       //Tính giá trị Page Server để so sánh
       #page_current_server := DINT_TO_UDINT(CEIL(UDINT_TO_REAL(#PageCurrentHMI) / 10));

       IF #page_current_server <> "DB_Machine".PageCurrentServerHistoricalPrevious THEN
           "DB_Server".PageHistorical.PageCurrent := #page_current_server;
           "DB_Server".ActionSearchLossHistorical := 1;
           "DB_Machine".PageCurrentServerHistoricalPrevious := #page_current_server;
       ELSE
           IF "DB_Server".ActionSearchLossHistorical = 2 OR "DB_Server".ActionSearchLossHistorical = 3 THEN
               //"ClearTableShowHMI"(2);
               "GetBufferHistoricalShowHMI"("DB_DataHMI".PageDataLossHistorical.PageCurrent);
           END_IF;
       END_IF;
   END_IF;
END_FUNCTION

// folder: Common

FUNCTION "IsIPAddress" : Bool   // FC1, SCL
TITLE = IsIPAddress
{ S7_Optimized_Access := 'TRUE' }
VERSION : 0.1
// Evaluates whether a given String contains a valid IP address
   VAR_INPUT
      address : String;   // Address to be evaluated
   END_VAR
   VAR_OUTPUT
      ipAddress : IP_V4;   // Parsed IP address if passed address is IP address
   END_VAR
   VAR_TEMP
      tempAddress : String;   // Passed address
      tempOctet : String;   // Current octet
      tempIndex : DInt;   // Index for loop
      tempPos : Int;   // Position of found separator
      tempNum : Int;   // Converted octet
      tempIp : IP_V4;   // Parsed IP address
   END_VAR
   // Ret_Val : Return value
   VAR CONSTANT
      MAX_VALUE : USInt := 255;   // Max. valid value of octet
      NUM_OCTETS : DInt := 4;   // Number of octets
      CHAR_ZERO : Char := '0';   // ASCII character '0'
   END_VAR
BEGIN
   REGION BLOCK INFO HEADER
     //===============================================================================
     // SIEMENS / (c)Copyright 2024
     //-------------------------------------------------------------------------------
     // Title:        IsIPAddress
     // Function:     Evaluates whether a given String contains a valid IP address
     // Library:      --
     // Author:       Siemens Industry Online Support
     // Tested with:  CPU 1515-2 PN V3.1
     // Engineering:  TIA Portal V17
     // Restrictions: --
     // Requirements: S7-1200 with firmware V4.4 or higher
     //               S7-1500 with firmware V2.0 or higher
     //-------------------------------------------------------------------------------
     // Change log table:
     // Version  | Date       | Expert in charge       | Changes applied
     //-------------------------------------------------------------------------------
     // 01.00.00 | 2024-02-12 | Online Support         | First released version
     //===============================================================================
   END_REGION

   #tempAddress := #address;
   #IsIPAddress := FALSE; // Will be overwritten if IP address is detected
   #ipAddress := #tempIp; // Zero output parameter

   FOR #tempIndex := 1 TO #NUM_OCTETS DO
     #tempPos := FIND(IN1 := #tempAddress, IN2 := '.'); // Find separator

     IF (#tempPos > 0 OR #tempIndex = #NUM_OCTETS) // Separator found with exception of last octet
       AND NOT (#tempPos > 0 AND #tempIndex = #NUM_OCTETS) // No separator found in last octet
       AND #tempPos <= 4 // 3  characters or less
     THEN
       IF #tempIndex < #NUM_OCTETS THEN // First three octets
         #tempOctet := LEFT(IN := #tempAddress, L := #tempPos - 1);
       ELSE// Last octet
         #tempOctet := #tempAddress;
       END_IF;

       STRG_VAL(IN := #tempOctet,
                FORMAT := 0,
                P := 1,
                OUT => #tempNum);

       IF #tempNum >= 0 AND #tempNum <= #MAX_VALUE // Within 0 and 255
         AND NOT (#tempNum = 0 AND #tempIndex = 1) // Not 0 in first octet
         AND NOT (#tempNum = 0 AND #tempOctet[1] <> #CHAR_ZERO) // Not 0 because of invalid character
       THEN
         #tempIp.ADDR[#tempIndex] := INT_TO_BYTE(#tempNum);
         #tempAddress := RIGHT(IN := #tempAddress, L := LEN(#tempAddress) - #tempPos); // Remove evaluated octet
       ELSE // Address is not IP address
         EXIT;
       END_IF;
     ELSE // Address is not IP address
       EXIT;
     END_IF;

     IF #tempIndex = #NUM_OCTETS THEN // End of loop reached, address is IP address
       #ipAddress := #tempIp;
       #IsIPAddress := true;
     END_IF;
   END_FOR;
END_FUNCTION

// folder: CommonFunctions

FUNCTION_BLOCK "InputFilter"   // FB4, LAD
{ S7_Optimized_Access := 'TRUE' }
VERSION : 0.1
   VAR_INPUT
      bInputTrigger : Bool;
      TonFilter_x1ms : Int := 10;   // x1ms
      ToffFilter_x1ms : Int := 10;   // x1ms
   END_VAR
   VAR_OUTPUT
      bOutput_P : Bool;
      bOutput_N : Bool;
   END_VAR
   VAR RETAIN
      P_tmp : Bool;
      N_tmp : Bool;
   END_VAR
   VAR
      Ton_start : Bool;
      Toff_start : Bool;
   END_VAR
   VAR RETAIN
      IEC_Ton : IEC_TIMER;
      IEC_Toff : IEC_TIMER;
   END_VAR
   VAR
      TimerTon : Time := T#10ms;
      TimerToff : Time := T#10ms;
   END_VAR
   VAR_TEMP   // added for the SCL form of the ladder/FBD networks
      _w1 : Bool;
   END_VAR
BEGIN

REGION Network 1
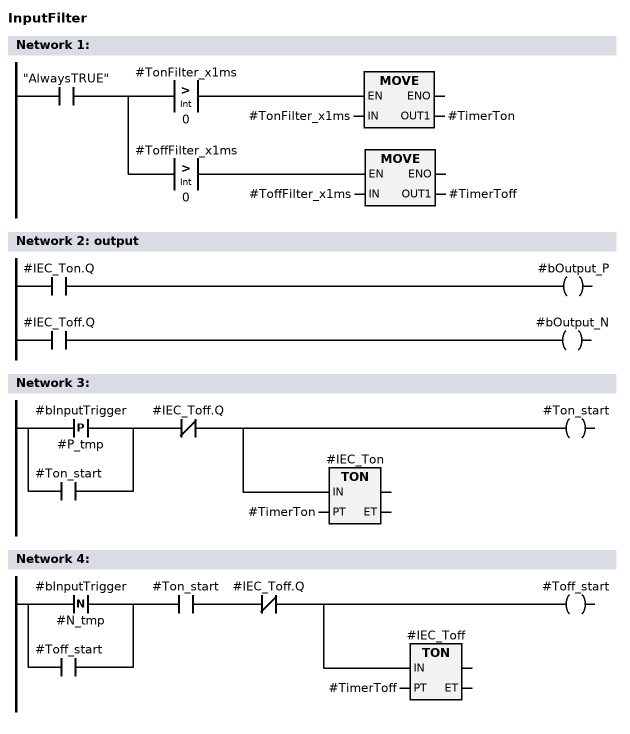
   RUNG wire#powerrail
      Contact( "AlwaysTRUE" )
      wire#w1
      { S7_Templates := "SrcType := Int" } GT_Contact(in1 := #TonFilter_x1ms, in2 := 0)
      Move(in := #TonFilter_x1ms, out1 => #TimerTon)
   END_RUNG
   RUNG wire#w1
      { S7_Templates := "SrcType := Int" } GT_Contact(in1 := #ToffFilter_x1ms, in2 := 0)
      Move(in := #ToffFilter_x1ms, out1 => #TimerToff)
   END_RUNG
   // the same network as SCL:
   IF "AlwaysTRUE" AND (#TonFilter_x1ms > 0) THEN #TimerTon := #TonFilter_x1ms; END_IF;
   IF "AlwaysTRUE" AND (#ToffFilter_x1ms > 0) THEN #TimerToff := #ToffFilter_x1ms; END_IF;
END_REGION

REGION Network 2: output
   RUNG wire#powerrail
      Contact( #IEC_Ton.Q )
      Coil( #bOutput_P )
   END_RUNG
   RUNG wire#powerrail
      Contact( #IEC_Toff.Q )
      Coil( #bOutput_N )
   END_RUNG
   // the same network as SCL:
   #bOutput_P := #IEC_Ton.Q;
   #bOutput_N := #IEC_Toff.Q;
END_REGION

REGION Network 3
   #_w1 := #bInputTrigger AND NOT #P_tmp;   // rising edge of #bInputTrigger
   #P_tmp := #bInputTrigger;
   #Ton_start := (#_w1 OR #Ton_start) AND NOT #IEC_Toff.Q;
   #IEC_Ton.TON(IN := #Ton_start, PT := #TimerTon);
END_REGION

REGION Network 4
   #_w1 := NOT #bInputTrigger AND #N_tmp;   // falling edge of #bInputTrigger
   #N_tmp := #bInputTrigger;
   #Toff_start := (#_w1 OR #Toff_start) AND #Ton_start AND NOT #IEC_Toff.Q;
   #IEC_Toff.TON(IN := #Toff_start, PT := #TimerToff);
END_REGION
END_FUNCTION_BLOCK

// folder: CommonFunctions/Analog

FUNCTION "AnalogScaling" : Void   // FC3, LAD
{ S7_Optimized_Access := 'TRUE' }
VERSION : 0.1
   VAR_INPUT
      AnalogInput : Int;   // Analog input as integer
      Lower : Real;   // Min - từ nhà sx
      Upper : Real;   // Max - từ nhà sx
      Min_Raw : Int;
      Max_Raw : Int;
   END_VAR
   VAR_OUTPUT
      ScaledOutput : Real;
   END_VAR
   VAR_TEMP
      normRealOutTmp : Real;
   END_VAR
BEGIN

REGION Network 1
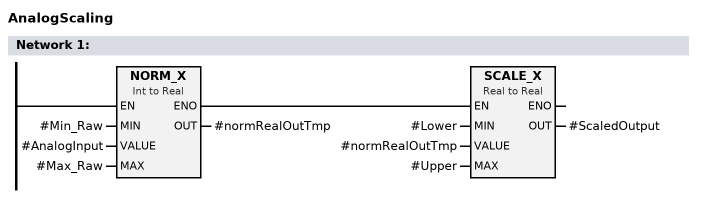
   RUNG wire#powerrail
      { S7_Templates := "[SrcType := Int, DestType := Real]" } Normalize(min := #Min_Raw, value := #AnalogInput, max := #Max_Raw, out => #normRealOutTmp)
      { S7_Templates := "[SrcType := Real, DestType := Real]" } Scale(min := #Lower, value := #normRealOutTmp, max := #Upper, out => #ScaledOutput)
   END_RUNG
   // the same network as SCL:
   #normRealOutTmp := NORM_X(MIN := #Min_Raw, VALUE := #AnalogInput, MAX := #Max_Raw);
   #ScaledOutput := SCALE_X(MIN := #Lower, VALUE := #normRealOutTmp, MAX := #Upper);
END_REGION
END_FUNCTION

FUNCTION "AnalogScallingWithFormatDigit" : Void   // FC5, LAD
{ S7_Optimized_Access := 'TRUE' }
VERSION : 0.1
   VAR_INPUT
      AnalogRawInput : Int;   // Analog input as integer
      Lower : Real;   // Min - từ nhà sx
      Upper : Real;   // Max - từ nhà sx
      Min_Raw : Int;
      Max_Raw : Int;
      Number_digit : Int;
   END_VAR
   VAR_OUTPUT
      RealOutput : Real;
      DintOutput : DInt;
   END_VAR
   VAR_TEMP
      scaleRealOutTmp : Real;
      normRealOutTmp : Real;
   END_VAR
   VAR_TEMP   // added for the SCL form of the ladder/FBD networks
      _w1 : Bool;
   END_VAR
BEGIN

REGION Network 1
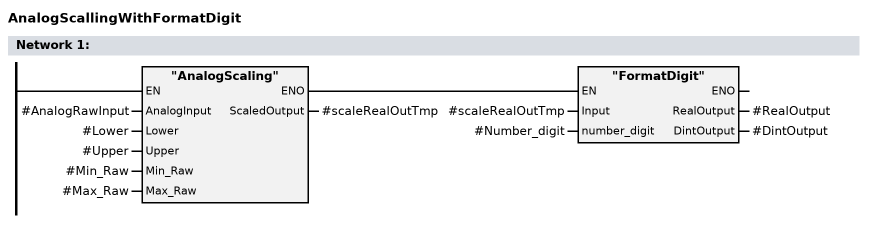
   RUNG wire#powerrail
      "AnalogScaling"(AnalogInput := #AnalogRawInput, Lower := #Lower, Upper := #Upper, Min_Raw := #Min_Raw, Max_Raw := #Max_Raw, ScaledOutput => #scaleRealOutTmp)
      "FormatDigit"(Input := #scaleRealOutTmp, number_digit := #Number_digit, RealOutput => #RealOutput, DintOutput => #DintOutput)
   END_RUNG
   // the same network as SCL:
   "AnalogScaling"(AnalogInput := #AnalogRawInput,
                   Lower := #Lower,
                   Upper := #Upper,
                   Min_Raw := #Min_Raw,
                   Max_Raw := #Max_Raw,
                   ScaledOutput => #scaleRealOutTmp,
                   ENO => #_w1);
   IF #_w1 THEN
       "FormatDigit"(Input := #scaleRealOutTmp,
                     number_digit := #Number_digit,
                     RealOutput => #RealOutput,
                     DintOutput => #DintOutput);
   END_IF;
END_REGION
END_FUNCTION

FUNCTION "CalculatorAxisYChart" : Void   // FC56, SCL
{ S7_Optimized_Access := 'TRUE' }
VERSION : 0.1
   VAR_INPUT
      Actual : DInt;
      Min : DInt;
      Max : DInt;
   END_VAR
   VAR_OUTPUT
      Min_AxisY : DInt;
      Max_AxisY : DInt;
   END_VAR
   VAR_TEMP
      value_min_temp : DInt;
      value_max_temp : DInt;
   END_VAR
   VAR CONSTANT
      OffsetMin : Real := 0.9;
      OffsetMax : Real := 1.1;
   END_VAR
BEGIN
   //Min Axits
   IF #Min < #Actual THEN
       #Min_AxisY := REAL_TO_DINT(DINT_TO_REAL(#Min) * #OffsetMin);
   ELSE
       #Min_AxisY := REAL_TO_DINT(DINT_TO_REAL(#Actual) * #OffsetMin);
   END_IF;


   //Max Axits
   IF #Max > #Actual THEN
       #Max_AxisY := ROUND_DINT(DINT_TO_REAL(#Max) * #OffsetMax);
   ELSE
       #Max_AxisY := ROUND_DINT(DINT_TO_REAL(#Actual) * #OffsetMax);
   END_IF;
END_FUNCTION

// folder: CommonFunctions/ClearBuffer

FUNCTION "ClearTableShowHMI" : Void   // FC37, SCL
{ S7_Optimized_Access := 'TRUE' }
VERSION : 0.1
   VAR_INPUT
      "1: table in shift, 2:table historical, 3: table spare part" : UInt;
   END_VAR
   VAR_TEMP
      index_for : USInt;
   END_VAR
BEGIN
   IF #"1: table in shift, 2:table historical, 3: table spare part" = 1  THEN
       FOR #index_for := 1 TO 5 DO
           "DB_DataHMI".DataLossInShiftShowHmiDTO[#index_for]."no." := 0;
           "DB_DataHMI".DataLossInShiftShowHmiDTO[#index_for].LossCode := 0;
           "DB_DataHMI".DataLossInShiftShowHmiDTO[#index_for].StartDateAsStr := '';
           "DB_DataHMI".DataLossInShiftShowHmiDTO[#index_for].StartTimeAsStr := '';
           "DB_DataHMI".DataLossInShiftShowHmiDTO[#index_for].EndDateAsStr := '';
           "DB_DataHMI".DataLossInShiftShowHmiDTO[#index_for].EndTimeAsStr := '';
           "DB_DataHMI".DataLossInShiftShowHmiDTO[#index_for].DurationAsStr := '';
           "DB_DataHMI".DataLossInShiftShowHmiDTO[#index_for].GroupLossReason := '';
           "DB_DataHMI".DataLossInShiftShowHmiDTO[#index_for].Description := '';
           "DB_DataHMI".DataLossInShiftShowHmiDTO[#index_for].IsHaveData := FALSE;
       END_FOR;
   ELSIF #"1: table in shift, 2:table historical, 3: table spare part" = 2  THEN
       FOR #index_for := 1 TO 5 DO
           "DB_DataHMI".DataLossHistoricalShowHmiDTO[#index_for]."no." := 0;
           "DB_DataHMI".DataLossHistoricalShowHmiDTO[#index_for].LossCode := 0;
           "DB_DataHMI".DataLossHistoricalShowHmiDTO[#index_for].StartDateAsStr := '';
           "DB_DataHMI".DataLossHistoricalShowHmiDTO[#index_for].StartTimeAsStr := '';
           "DB_DataHMI".DataLossHistoricalShowHmiDTO[#index_for].EndDateAsStr := '';
           "DB_DataHMI".DataLossHistoricalShowHmiDTO[#index_for].EndTimeAsStr := '';
           "DB_DataHMI".DataLossHistoricalShowHmiDTO[#index_for].DurationAsStr := '';
           "DB_DataHMI".DataLossHistoricalShowHmiDTO[#index_for].GroupLossReason := '';
           "DB_DataHMI".DataLossHistoricalShowHmiDTO[#index_for].Description := '';
           "DB_DataHMI".DataLossHistoricalShowHmiDTO[#index_for].IsHaveData := FALSE;
       END_FOR;
   ELSIF #"1: table in shift, 2:table historical, 3: table spare part" = 3  THEN
       FOR #index_for := 1 TO 5 DO
           "DB_DataHMI".DataSparePartShowHmiDTO[#index_for]."No." := 0;
           "DB_DataHMI".DataSparePartShowHmiDTO[#index_for].Name := '';
           "DB_DataHMI".DataSparePartShowHmiDTO[#index_for].ProductCount := 0;
           "DB_DataHMI".DataSparePartShowHmiDTO[#index_for].StartTime := '';
           "DB_DataHMI".DataSparePartShowHmiDTO[#index_for].EndTime := '';
           "DB_DataHMI".DataSparePartShowHmiDTO[#index_for].IsHaveData := FALSE;
       END_FOR;
   END_IF;
END_FUNCTION

FUNCTION "ClearBufferLossInShift" : Void   // FC41, SCL
{ S7_Optimized_Access := 'TRUE' }
VERSION : 0.1
   VAR_TEMP
      index_for : USInt;
   END_VAR
BEGIN
   FOR #index_for := 1 TO 100 DO
       "BuffersLoss_DB".buffer_loss_in_shift[#index_for].id := 0;
       "BuffersLoss_DB".buffer_loss_in_shift[#index_for].losscode := 0;
       "BuffersLoss_DB".buffer_loss_in_shift[#index_for].statusServer := 0;
   END_FOR;
   "GLobalDB_LossManagementDB".index_buffer_loss_in_shift_current := 1;
   "GLobalDB_LossManagementDB".id_loss := 1;
   "DB_DataHMI".TotalDataInShift := 0;
   "DB_Machine".NumberLossInShift := 0;

   "DB_DataHMI".PageDataLossInShift.PageCurrent := 1;
   "DB_DataHMI".PageDataLossInShift.MaxPage := 1;
   "DB_DataHMI".PageDataLossInShift.TotalData := 0;
END_FUNCTION

FUNCTION "ClearBufferStatusMachineOfServer" : Void   // FC55, SCL
{ S7_Optimized_Access := 'TRUE' }
VERSION : 0.1
   VAR_TEMP
      index_for : USInt;
   END_VAR
BEGIN
   "StatusMachineSendServerDB".index_current := 1;

   FOR #index_for := 1 TO 50 DO
       "StatusMachineSendServerDB".StatusMachineBuffer[#index_for].time_start.YEAR := 2000;
       "StatusMachineSendServerDB".StatusMachineBuffer[#index_for].time_start.MONTH := 1;
       "StatusMachineSendServerDB".StatusMachineBuffer[#index_for].time_start.DAY := 1;

       "StatusMachineSendServerDB".StatusMachineBuffer[#index_for].timer_end.YEAR := 2000;
       "StatusMachineSendServerDB".StatusMachineBuffer[#index_for].timer_end.MONTH := 1;
       "StatusMachineSendServerDB".StatusMachineBuffer[#index_for].timer_end.DAY := 1;
   END_FOR;
END_FUNCTION

FUNCTION "BufferLossReasonGroupDefault" : Void   // FC57, SCL
{ S7_Optimized_Access := 'TRUE' }
VERSION : 0.1
   VAR_TEMP
      index_for : UInt;
   END_VAR
BEGIN
   FOR #index_for := 1 TO 10 DO
       "SettingsDB_LossDescription".loss_name_group[#index_for] := CONCAT(IN1 := 'Group:', IN2 := UINT_TO_STRING(#index_for));
   END_FOR;


   FOR #index_for := 1 TO 100 DO
       "SettingsDB_LossDescription".loss_descriptions[#index_for].description := CONCAT(IN1 := 'Reason:', IN2 := UINT_TO_STRING(#index_for));
       "SettingsDB_LossDescription".loss_descriptions[#index_for].group_id := #index_for MOD 10;
   END_FOR;


   "SettingsDB_LossDescription".number_loss_reason := 100;
END_FUNCTION

FUNCTION "ClearBufferTempLossInShift" : Void   // FC65, SCL
{ S7_Optimized_Access := 'TRUE' }
VERSION : 0.1
   VAR_TEMP
      i : USInt;
   END_VAR
BEGIN
   FOR #i := 1 TO 100 DO
       "DB_Machine".buffer_index_sort[#i].id := 0;
       "DB_Machine".buffer_index_sort[#i].index_buffer := 0;
   END_FOR;
END_FUNCTION

FUNCTION "ClearBufferLossHistorical" : Void   // FC68, SCL
{ S7_Optimized_Access := 'TRUE' }
VERSION : 0.1
   VAR_TEMP
      index_for : USInt;
   END_VAR
BEGIN
   FOR #index_for := 1 TO 50 DO
       "BuffersLoss_DB".buffer_loss_in_historical[#index_for].id := 0;
       "BuffersLoss_DB".buffer_loss_in_historical[#index_for].losscode := 0;
       "BuffersLoss_DB".buffer_loss_in_historical[#index_for].statusServer := 0;
       "BuffersLoss_DB".buffer_loss_in_historical[#index_for].duration := 0;
   END_FOR;

   "DB_Server".PageHistorical.TotalData := 0;
   "DB_Server".PageHistorical.MaxPage := 1;
   "DB_Server".PageHistorical.PageCurrent := 1;
   "DB_Server".TotalDurationPageHistorical := 0;
END_FUNCTION

FUNCTION "ClearBufferSparePart" : Void   // FC70, SCL
{ S7_Optimized_Access := 'TRUE' }
VERSION : 0.1
   VAR_TEMP
      index_for : USInt;
   END_VAR
BEGIN
   FOR #index_for := 1 TO 30 DO
       "BufferServerSend".buffer_spare_part[#index_for].name := '';
       "BufferServerSend".buffer_spare_part[#index_for].product_count := 0;
   END_FOR;

   "DB_Server".PageDataSparePart.TotalData := 0;
   "DB_Server".PageDataSparePart.MaxPage := 1;
   "DB_Server".PageDataSparePart.PageCurrent := 1;
END_FUNCTION

FUNCTION "ResetCheckBoxLossReason" : Void   // FC71, SCL
{ S7_Optimized_Access := 'TRUE' }
VERSION : 0.1
   VAR_TEMP
      index : USInt;
   END_VAR
BEGIN
   FOR #index := 1 TO 10 DO
       "DB_DataHMI".CheckboxLossReason[#index] := 0;
   END_FOR;
END_FUNCTION

FUNCTION "ResetCheckBoxLossGroup" : Void   // FC72, SCL
{ S7_Optimized_Access := 'TRUE' }
VERSION : 0.1
   VAR_TEMP
      index : USInt;
   END_VAR
BEGIN
   FOR #index := 1 TO 10 DO
       "DB_DataHMI".CheckboxLossGroup[#index] := 0;
   END_FOR;
END_FUNCTION

FUNCTION "ResetArraySpeedTemp" : Void   // FC73, SCL
{ S7_Optimized_Access := 'TRUE' }
VERSION : 0.1
   VAR_TEMP
      index : USInt;
   END_VAR
BEGIN
   FOR #index := 1 TO 50 DO
       "SensorSpeed_DB".array_speed_temp[#index] := 0;
   END_FOR;
END_FUNCTION

// folder: CommonFunctions/Math

FUNCTION "FormatDigit" : Void   // FC4, LAD
{ S7_Optimized_Access := 'TRUE' }
VERSION : 0.1
   VAR_INPUT
      Input : Real;
      number_digit : Int;
   END_VAR
   VAR_OUTPUT
      RealOutput : Real;
      DintOutput : DInt;
   END_VAR
   VAR_TEMP
      dint_tmp : DInt;
      real_tmp : Real;
      tmp_1 : DInt;
      tmp_2 : DInt;
      real_tmp_1 : Real;
      dint_tmp_2 : DInt;
   END_VAR
BEGIN

REGION Network 1
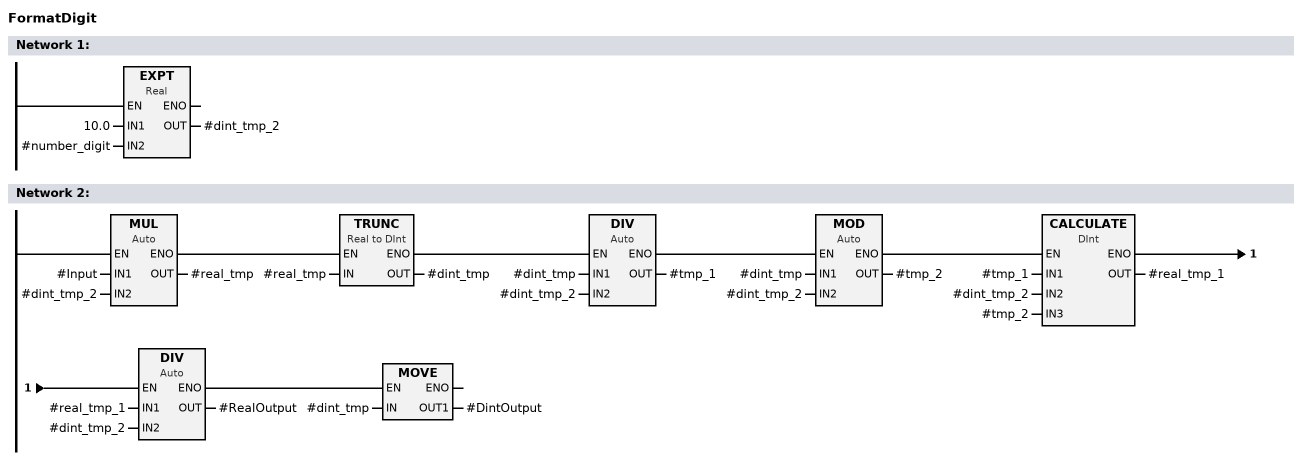
   #dint_tmp_2 := 10.0 ** #number_digit;
END_REGION

REGION Network 2
   RUNG wire#powerrail
      Mul(in1 := #Input, in2 := #dint_tmp_2, out => #real_tmp)
      { S7_Templates := "[SrcType := Real, DestType := DInt]" } Trunc(in := #real_tmp, out => #dint_tmp)
      Div(in1 := #dint_tmp, in2 := #dint_tmp_2, out => #tmp_1)
      Mod(in1 := #dint_tmp, in2 := #dint_tmp_2, out => #tmp_2)
      { S7_Templates := "SrcType := DInt"; S7_Expression := "(IN1 * IN2 + IN3)" } Calculate(in1 := #tmp_1, in2 := #dint_tmp_2, in3 := #tmp_2, out => #real_tmp_1)
      Div(in1 := #real_tmp_1, in2 := #dint_tmp_2, out => #RealOutput)
      Move(in := #dint_tmp, out1 => #DintOutput)
   END_RUNG
   // the same network as SCL:
   #real_tmp := #Input * #dint_tmp_2;
   #dint_tmp := TRUNC(#real_tmp);
   #tmp_1 := #dint_tmp / #dint_tmp_2;
   #tmp_2 := #dint_tmp MOD #dint_tmp_2;
   #real_tmp_1 := (#tmp_1 * #dint_tmp_2 + #tmp_2);
   #RealOutput := #real_tmp_1 / #dint_tmp_2;
   #DintOutput := #dint_tmp;
END_REGION
END_FUNCTION

FUNCTION "Avg_Real" : Void   // FC10, SCL
{ S7_Optimized_Access := 'TRUE' }
VERSION : 0.1
   VAR_INPUT
      "IN 1" : Real;
      "IN 2" : Real;
      "IN 3" : Real;
   END_VAR
   VAR_OUTPUT
      Out : Real;
   END_VAR
BEGIN
   #Out := (#"IN 1" + #"IN 2" + #"IN 3") / 3;
END_FUNCTION

FUNCTION "Avg_Dint" : Void   // FC11, SCL
{ S7_Optimized_Access := 'TRUE' }
VERSION : 0.1
   VAR_INPUT
      "IN 1" : DInt;
      "IN 2" : DInt;
      "IN 3" : DInt;
   END_VAR
   VAR_OUTPUT
      Out : DInt;
   END_VAR
BEGIN
   #Out := (#"IN 1" + #"IN 2" + #"IN 3") / 3;
END_FUNCTION

FUNCTION "CompareDTL" : Void   // FC64, SCL
{ S7_Optimized_Access := 'TRUE' }
VERSION : 0.1
   VAR_INPUT
      DTL_Input1 : DTL;
      DTL_Input2 : DTL;
   END_VAR
   VAR_OUTPUT
      Result : Bool;
   END_VAR
BEGIN
   IF #DTL_Input1.YEAR=#DTL_Input2.YEAR AND
       #DTL_Input1.MONTH=#DTL_Input2.MONTH AND
       #DTL_Input1.DAY=#DTL_Input2.DAY AND
       #DTL_Input1.HOUR=#DTL_Input2.HOUR AND
       #DTL_Input1.MINUTE=#DTL_Input2.MINUTE AND
       #DTL_Input1.SECOND=#DTL_Input2.SECOND THEN
       #Result := TRUE;
   ELSE
       #Result := FALSE;
   END_IF;
END_FUNCTION

// folder: CommonFunctions/String

FUNCTION "DTL_to_String" : Void   // FC7, SCL
{ S7_Optimized_Access := 'TRUE' }
VERSION : 0.1
   VAR_INPUT
      DTL : DTL;
   END_VAR
   VAR_OUTPUT
      OutputStr : String;
   END_VAR
   VAR_TEMP
      year : String;
      month : String;
      day : String;
      hour : String;
      minute : String;
      second : String;
   END_VAR
BEGIN
   #OutputStr := "LGF_DTLToString_ISO"("date":=#DTL, separator:='/');
END_FUNCTION

FUNCTION "Trim" : Void   // FC8, SCL
{ S7_Optimized_Access := 'TRUE' }
VERSION : 0.1
   VAR_INPUT
      InputStr : String;
   END_VAR
   VAR_OUTPUT
      OutputStr : String;
   END_VAR
   VAR_TEMP
      Leng : Int;
      Cnt : Int;
      Index : USInt;
   END_VAR
BEGIN
   #Leng := LEN(#InputStr);
   #Index := 0;
   #OutputStr := '';
   FOR #Cnt := 0 TO #Leng DO
       IF #InputStr[#Cnt] <> ' ' THEN
           #OutputStr[#Index] := #InputStr[#Cnt];
           #Index := #Index + 1;
       END_IF;
   END_FOR;
END_FUNCTION

FUNCTION "TimeToString" : Void   // FC9, SCL
{ S7_Optimized_Access := 'TRUE' }
VERSION : 0.1
   VAR_INPUT
      timeValue : Time;
   END_VAR
   VAR_OUTPUT
      OutputStr : String;
   END_VAR
   VAR_TEMP
      day : String;
      hour : String;
      minute : String;
      second : String;
      milisecond : String;
      output_str : String;
      aaa : Int;
      bbb : Char;
      tempTimeMilliseconds : DInt;   // Temp integer to calculate the different time values
      tempDays : DInt;   // Temp number for days
      tempHours : DInt;   // Temp number for hours
      tempMinutes : DInt;   // Temp number for minutes
      tempSecond : DInt;   // Temp number for seconds
      tempMillisecond : DInt;   // Temp number for milliseconds
   END_VAR
   VAR CONSTANT
      MS_PER_DAY : DInt := 86400000;   // Milliseconds per day
      MS_PER_HOUR : DInt := 3600000;   // Milliseconds per hour
      MS_PER_MINUTE : DInt := 60000;   // Milliseconds per minute
      MS_PER_SECOND : DInt := 1000;   // Milliseconds per second
      NUMBER_OF_CHAR_TO_DEL : Int := 1;   // Number of characters to be deleted
      FIRST_POSITION : Int := 1;   // Position in string from where the deletion will be begin
      NO_REMAINDER : Int := 0;   // Remainder from devision
   END_VAR
BEGIN
   // convert from time to millisecond
   #tempTimeMilliseconds := TIME_TO_DINT(#timeValue);

   // calculate the days and remaining hours
   #tempDays := #tempTimeMilliseconds / #MS_PER_DAY;
   #tempTimeMilliseconds := #tempTimeMilliseconds MOD #MS_PER_DAY;

   // calculate the hours and remaining minutes
   #tempHours := #tempTimeMilliseconds / #MS_PER_HOUR;
   #tempTimeMilliseconds := #tempTimeMilliseconds MOD #MS_PER_HOUR;

   // calculate the minutes and remaining seconds
   #tempMinutes := #tempTimeMilliseconds / #MS_PER_MINUTE;
   #tempTimeMilliseconds := #tempTimeMilliseconds MOD #MS_PER_MINUTE;

   // calculate the seconds and remaining milliseconds
   #tempSecond := #tempTimeMilliseconds / #MS_PER_SECOND;
   #tempMillisecond := #tempTimeMilliseconds MOD #MS_PER_SECOND;

   IF (#tempSecond > 10) THEN
       #second := DINT_TO_STRING(#tempSecond);
       #second := RIGHT(IN := #second, L := 2);
       #second := CONCAT(IN1 := #second, IN2 := 'S');
   ELSE
       IF (#tempSecond > 0) THEN
           #second := DINT_TO_STRING(#tempSecond);
           #second := RIGHT(IN := #second, L := 1);
           #second := CONCAT(IN1 := '0', IN2 := #second, IN3 := 'S');
       ELSE
           #second := '00S';
       END_IF;
   END_IF;

   IF (#tempMinutes > 10) THEN
       #minute := DINT_TO_STRING(#tempMinutes);
       #minute := RIGHT(IN := #minute, L := 2);
       #minute := CONCAT(IN1 := #minute, IN2 := 'M:');
   ELSE
       IF (#tempMinutes > #NO_REMAINDER) THEN
           #minute := DINT_TO_STRING(#tempMinutes);
           #minute := RIGHT(IN := #minute, L := 1);
           #minute := CONCAT(IN1 := '0', IN2 := #minute, IN3 := 'M:');
       END_IF;
   END_IF;

   IF (#tempHours > 10) THEN
       #hour := DINT_TO_STRING(#tempHours);
       #hour := RIGHT(IN := #hour, L := 2);
       #hour := CONCAT(IN1 := #hour, IN2 := 'H:');
   ELSE
       IF (#tempHours > #NO_REMAINDER) THEN
           #hour := DINT_TO_STRING(#tempHours);
           #hour := RIGHT(IN := #hour, L := 1);
           #hour := CONCAT(IN1 := '0', IN2 := #hour, IN3 := 'H:');
       END_IF;
   END_IF;

   // IF (#tempDays > #NO_REMAINDER) THEN
   //     #day := DINT_TO_STRING(#tempDays);
   //     //#day := RIGHT(IN := #hour, L := 2);
   //     #day := CONCAT(IN1 := #day, IN2 := 'D:');
   // END_IF;

   IF (#tempDays > 10) THEN
       #day := DINT_TO_STRING(#tempDays);
       #day := RIGHT(IN := #day, L := 2);
       #day := CONCAT(IN1 := #day, IN2 := 'M:');
   ELSE
       IF (#tempDays > #NO_REMAINDER) THEN
           #day := DINT_TO_STRING(#tempDays);
           #day := RIGHT(IN := #day, L := 1);
           #day := CONCAT(IN1 := #day, IN2 := 'D:');
       END_IF;
   END_IF;



   //#output_str := "LGF_TimeToString"(timeValue := #timeValue, stringDay => #day, stringHour => #hour, stringMinute => #minute, stringSecond => #second, stringMilliSecond => #milisecond);
   // "Trim"(InputStr := #day,OutputStr=>#day);
   // "Trim"(InputStr := #hour,OutputStr => #hour);
   // "Trim"(InputStr := #minute,OutputStr => #minute);
   // "Trim"(InputStr := #second,OutputStr => #second);
   // "Trim"(InputStr := #day,OutputStr => #day);

   // #bbb := RIGHT(IN:=#minute, L:=1);
   // #aaa := STRING_TO_INT(#minute);

   // IF LEN(#day) = 1 THEN
   //     #day := CONCAT(IN1 := '0', IN2 := #day, IN3 := 'D_');
   // ELSE
   //     IF LEN(#day) = 2 THEN
   //         #day := CONCAT(IN1 := #day, IN2 := 'D_');
   //     END_IF;
   // END_IF;

   // IF LEN(#hour) = 1 THEN
   //     #hour := CONCAT(IN1 := '0', IN2 := #hour, IN3 := 'H_');
   // ELSE
   //     IF LEN(#hour) = 2 THEN
   //         #hour := CONCAT(IN1 := #hour, IN2 := 'H_');
   //     END_IF;
   // END_IF;

   // IF LEN(#minute) = 1 THEN
   //     #minute := CONCAT(IN1 := '0', IN2 := #minute, IN3 := 'M_');
   // ELSE
   //     IF LEN(#minute) = 2 THEN
   //         #minute := CONCAT(IN1 := #minute, IN2 := 'M_');
   //     END_IF;
   // END_IF;

   // IF LEN(#second) = 1 THEN
   //     #second := CONCAT(IN1 := '0', IN2 := #second, IN3 := 'S');
   // ELSE
   //     IF LEN(#second) = 2 THEN
   //         #second := CONCAT(IN1 := #second, IN2 := 'S');
   //     END_IF;
   // END_IF;
   #OutputStr := CONCAT(IN1 := #day,
                        IN2 := #hour,
                        IN3 := #minute,
                        IN4 := #second);
END_FUNCTION

FUNCTION "DTL_to_DateString" : Void   // FC34, SCL
{ S7_Optimized_Access := 'TRUE' }
VERSION : 0.1
   VAR_INPUT
      DTL : DTL;
   END_VAR
   VAR_OUTPUT
      DateTimeString : String;
   END_VAR
   VAR_TEMP
      Year : UInt;
      StrYear : String;
      StrMonth : String;
      StrDay : String;
   END_VAR
BEGIN

   IF #DTL.YEAR>=2000 THEN
       "FC_Trim"(InputStr := UINT_TO_STRING(#DTL.YEAR),
                 OutputStr => #StrYear);

       "FC_Trim"(InputStr := USINT_TO_STRING(#DTL.MONTH),
                 OutputStr => #StrMonth);

       "FC_Trim"(InputStr := USINT_TO_STRING(#DTL.DAY),
                 OutputStr => #StrDay);

       IF LEN(#StrMonth) < 2 THEN
           #StrMonth := CONCAT(IN1 := '0', IN2 := #StrMonth);
       END_IF;
       IF LEN(#StrDay) < 2 THEN
           #StrDay := CONCAT(IN1 := '0', IN2 := #StrDay);
       END_IF;

       #DateTimeString := CONCAT(IN1 := #StrYear,
                                 IN2 := '-',
                                 IN3 := #StrMonth,
                                 IN4 := '-',
                                 IN5 := #StrDay);
   ELSE
       #DateTimeString := '--/--/--/';
   END_IF;
END_FUNCTION

FUNCTION "DTL_to_TimeString" : Void   // FC35, SCL
{ S7_Optimized_Access := 'TRUE' }
VERSION : 0.1
   VAR_INPUT
      DTL : DTL;
   END_VAR
   VAR_OUTPUT
      DateTimeString : String;
   END_VAR
   VAR_TEMP
      StrHour : String;
      StrMinute : String;
      StrSecond : String;
   END_VAR
BEGIN
   "FC_Trim"(InputStr := USINT_TO_STRING(#DTL.HOUR),
             OutputStr => #StrHour);

   "FC_Trim"(InputStr := USINT_TO_STRING(#DTL.MINUTE),
             OutputStr => #StrMinute);

   "FC_Trim"(InputStr := USINT_TO_STRING(#DTL.SECOND),
             OutputStr => #StrSecond);

   IF LEN(#StrHour) < 2 THEN
       #StrHour := CONCAT(IN1 := '0', IN2 := #StrHour);
   END_IF;
   IF LEN(#StrMinute) < 2 THEN
       #StrMinute := CONCAT(IN1 := '0', IN2 := #StrMinute);
   END_IF;
   IF LEN(#StrSecond) < 2 THEN
       #StrSecond := CONCAT(IN1 := '0', IN2 := #StrSecond);
   END_IF;

   #DateTimeString := CONCAT(IN1 := #StrHour,
                             IN2 := ':',
                             IN3 := #StrMinute,
                             IN4 := ':',
                             IN5 := #StrSecond);
END_FUNCTION

FUNCTION "FC_Trim" : Void   // FC36, SCL
{ S7_Optimized_Access := 'TRUE' }
VERSION : 0.1
   VAR_INPUT
      InputStr : String;
   END_VAR
   VAR_OUTPUT
      OutputStr : String;
   END_VAR
   VAR_TEMP
      Leng : Int;
      index_for : Int;
      Index : USInt;
   END_VAR
BEGIN
   #Leng := LEN(#InputStr);
   #Index := 0;
   #OutputStr := '';
   FOR #index_for := 0 TO #Leng DO
       IF #InputStr[#index_for] <> ' ' AND #InputStr[#index_for] <> '+' THEN
           #OutputStr[#Index] := #InputStr[#index_for];
           #Index += 1;
       END_IF;
   END_FOR;
END_FUNCTION

FUNCTION "Cvt_Duration_to_String" : Void   // FC38, LAD
{ S7_Optimized_Access := 'TRUE' }
VERSION : 0.1
   VAR_INPUT
      "Time(ms)" : UDInt;
   END_VAR
   VAR_OUTPUT
      ConvertTimeToStr : String;
   END_VAR
   VAR_TEMP
      Hour : UInt;
      Minute : UInt;
      Second : UInt;
      StrHour : String;
      StrMinute : String;
      StrSecond : String;
   END_VAR
BEGIN

REGION Network 1: Đổi ms sang HH MM SS
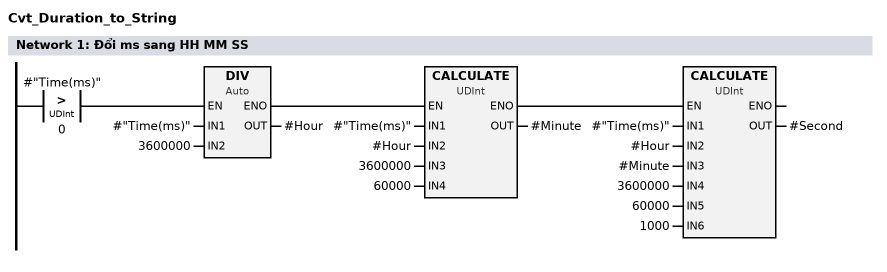
   RUNG wire#powerrail
      { S7_Templates := "SrcType := UDInt" } GT_Contact(in1 := #"Time(ms)", in2 := 0)
      Div(in1 := #"Time(ms)", in2 := 3600000, out => #Hour)
      { S7_Templates := "SrcType := UDInt"; S7_Expression := "(IN1-IN2*IN3)/IN4" } Calculate(in1 := #"Time(ms)", in2 := #Hour, in3 := 3600000, in4 := 60000, out => #Minute)
      { S7_Templates := "SrcType := UDInt"; S7_Expression := "(IN1-IN2*IN4-IN3*IN5)/IN6" } Calculate(in1 := #"Time(ms)", in2 := #Hour, in3 := #Minute, in4 := 3600000, in5 := 60000, in6 := 1000, out => #Second)
   END_RUNG
   // the same network as SCL:
   IF #"Time(ms)" > 0 THEN
       #Hour := #"Time(ms)" / 3600000;
       #Minute := (#"Time(ms)"-#Hour*3600000)/60000;
       #Second := (#"Time(ms)"-#Hour*3600000-#Minute*60000)/1000;
   END_IF;
END_REGION

REGION Network 2 (SCL): Chuyển sang string
   IF #"Time(ms)">0 THEN
       "FC_Trim"(InputStr := UINT_TO_STRING(#Hour),
                 OutputStr => #StrHour);
       "FC_Trim"(InputStr := UINT_TO_STRING(#Minute),
                 OutputStr => #StrMinute);
       "FC_Trim"(InputStr := UINT_TO_STRING(#Second),
                 OutputStr => #StrSecond);

       IF LEN(#StrHour) < 2 THEN
           #StrHour := CONCAT(IN1 := '0', IN2 := #StrHour);
       END_IF;
       IF LEN(#StrMinute) < 2 THEN
           #StrMinute := CONCAT(IN1 := '0', IN2 := #StrMinute);
       END_IF;
       IF LEN(#StrSecond) < 2 THEN
           #StrSecond := CONCAT(IN1 := '0', IN2 := #StrSecond);
       END_IF;

       #ConvertTimeToStr := CONCAT(IN1 := #StrHour,
                                 IN2 := ':',
                                 IN3 := #StrMinute,
                                 IN4 := ':',
                                 IN5 := #StrSecond);
   ELSE
       #ConvertTimeToStr := '00:00:00';
   END_IF;
END_REGION
END_FUNCTION

FUNCTION "DTL_to_StringV2" : Void   // FC51, SCL
{ S7_Optimized_Access := 'TRUE' }
VERSION : 0.1
   VAR_INPUT
      DTL : DTL;
   END_VAR
   VAR_OUTPUT
      DateTimeString : String;
   END_VAR
   VAR_TEMP
      Year : UInt;
      StrYear : String;
      StrMonth : String;
      StrDay : String;
      StrHour : String;
      StrMinute : String;
      StrSecond : String;
   END_VAR
BEGIN
   IF #DTL.YEAR >= 2000 THEN
       "FC_Trim"(InputStr := UINT_TO_STRING(#DTL.YEAR),
                 OutputStr => #StrYear);

       "FC_Trim"(InputStr := USINT_TO_STRING(#DTL.MONTH),
                 OutputStr => #StrMonth);

       "FC_Trim"(InputStr := USINT_TO_STRING(#DTL.DAY),
                 OutputStr => #StrDay);

       "FC_Trim"(InputStr := USINT_TO_STRING(#DTL.HOUR),
                 OutputStr => #StrHour);

       "FC_Trim"(InputStr := USINT_TO_STRING(#DTL.MINUTE),
                 OutputStr => #StrMinute);

       "FC_Trim"(InputStr := USINT_TO_STRING(#DTL.SECOND),
                 OutputStr => #StrSecond);


       IF LEN(#StrMonth) < 2 THEN
           #StrMonth := CONCAT(IN1 := '0', IN2 := #StrMonth);
       END_IF;
       IF LEN(#StrDay) < 2 THEN
           #StrDay := CONCAT(IN1 := '0', IN2 := #StrDay);
       END_IF;

       IF LEN(#StrHour) < 2 THEN
           #StrHour := CONCAT(IN1 := '0', IN2 := #StrHour);
       END_IF;
       IF LEN(#StrMinute) < 2 THEN
           #StrMinute := CONCAT(IN1 := '0', IN2 := #StrMinute);
       END_IF;
       IF LEN(#StrSecond) < 2 THEN
           #StrSecond := CONCAT(IN1 := '0', IN2 := #StrSecond);
       END_IF;

       #DateTimeString := CONCAT(IN1 := #StrYear,
                                 IN2 := '-',
                                 IN3 := #StrMonth,
                                 IN4 := '-',
                                 IN5 := #StrDay,
                                 IN6 := ' ',
                                 IN7 := #StrHour,
                                 IN8 := ':',
                                 IN9 := #StrMinute,
                                 IN10 := ':',
                                 IN11 := #StrSecond);
   ELSE
       #DateTimeString := '--/--/--';
   END_IF;
END_FUNCTION

FUNCTION "LGF_TimeToString" : String   // FC10043, SCL
TITLE = LGF_TimeToString
{ S7_Optimized_Access := 'TRUE' }
AUTHOR : Siemens_Digital_Industry
FAMILY : LGF
NAME : LGF_TimeToString
// This function converts a variable of the system data type `Time` into a variable of the data type `String`.
   VAR_INPUT
      timeValue : Time;   // Time value to convert Example: `T#1D_3H_45M_6S`
   END_VAR
   VAR_OUTPUT
      stringDay : String;   // Converted day as string
      stringHour : String;   // Converted hour as string
      stringMinute : String;   // Converted minute as string
      stringSecond : String;   // Converted second as string
      stringMilliSecond : String;   // Converted millisecond as string
   END_VAR
   VAR_TEMP
      tempTimeResult : String;   // Temp string to concat the results of conversions
      tempTimeMilliseconds : DInt;   // Temp integer to calculate the different time values
      tempDays : DInt;   // Temp number for days
      tempHours : DInt;   // Temp number for hours
      tempMinutes : DInt;   // Temp number for minutes
      tempSecond : DInt;   // Temp number for seconds
      tempMillisecond : DInt;   // Temp number for milliseconds
   END_VAR
   // Ret_Val : Converted time as string. Example: `1D3H45M6S0MS`
   VAR CONSTANT
      MS_PER_DAY : DInt := 86400000;   // Milliseconds per day
      MS_PER_HOUR : DInt := 3600000;   // Milliseconds per hour
      MS_PER_MINUTE : DInt := 60000;   // Milliseconds per minute
      MS_PER_SECOND : DInt := 1000;   // Milliseconds per second
      NUMBER_OF_CHAR_TO_DEL : Int := 1;   // Number of characters to be deleted
      FIRST_POSITION : Int := 1;   // Position in string from where the deletion will be begin
      NO_REMAINDER : Int := 0;   // Remainder from devision
   END_VAR
BEGIN
   REGION BLOCK INFO HEADER
     //===============================================================================
     // SIEMENS AG / (c)Copyright 2017
     //-------------------------------------------------------------------------------
     // Title:            LGF_TimeToString
     // Comment/Function: This function converts a time value to a string
     //                   When more than one time unit is specified, the value must not exceed 24 days, 23 hours, 59 minutes, 59 seconds or 999 milliseconds.
     //                   Output format is the folowing := '10D20H30M20S630MS', just existing parts would be added to the string
     // Library/Family:   LGF(Library General Functions)
     // Author:           Siemens Digital Industry Support
     // Tested with:      S7-PLCSIM Advanced V2.0 SP1
     // Engineering:      TIA Portal V14 SP1 Upd 5
     // Restrictions:     ENO mechanism is not used, no error handling
     // Requirements:     PLC (S7-1200 / S7-1500)
     //-------------------------------------------------------------------------------
     // Change log table:
     // Version  | Date       | Expert in charge       | Changes applied
     //----------|------------|------------------------|------------------------------
     // 01.00.00 | 03.07.2018 | Siemens Industry Online Support
     //                         First released version
     // 01.00.01 | 17.08.2018 | Siemens Industry Online Support
     //                         Upgrade: TIA V15 Update 2
     // 01.00.02 | 23.11.2018 | Siemens Industry Online Support
     //                         Upgrade: TIA V15.1
     // 01.00.03 | 02.07.2019 | Simatic Systems Support
     //                         Standard header and block parameters update, status parameter added
     // 01.00.05 | 09.07.2019 | Simatic Systems Support
     //                         Further improvements minimization and commends added
     // 01.00.06 | 30.07.2019 | Simatic Systems Support
     //                         Add ENO handling
     // 03.00.00 | 23.04.2020 | Simatic Systems Support | Set version to V3.0.0
     //                         Harmonize the version of the whole library
     // 03.00.01 | 23.02.2021 | Simatic Systems Support
     //                         Insert documentation
     //===============================================================================
   END_REGION Block info header

   REGION INITIALISATION
     #tempTimeResult := '';
   END_REGION

   REGION CONVERT
     // convert from time to millisecond
     #tempTimeMilliseconds := TIME_TO_DINT(#timeValue);

     // calculate the days and remaining hours
     #tempDays := #tempTimeMilliseconds / #MS_PER_DAY;
     #tempTimeMilliseconds := #tempTimeMilliseconds MOD #MS_PER_DAY;

     // calculate the hours and remaining minutes
     #tempHours := #tempTimeMilliseconds / #MS_PER_HOUR;
     #tempTimeMilliseconds := #tempTimeMilliseconds MOD #MS_PER_HOUR;

     // calculate the minutes and remaining seconds
     #tempMinutes := #tempTimeMilliseconds / #MS_PER_MINUTE;
     #tempTimeMilliseconds := #tempTimeMilliseconds MOD #MS_PER_MINUTE;

     // calculate the seconds and remaining milliseconds
     #tempSecond := #tempTimeMilliseconds / #MS_PER_SECOND;
     #tempMillisecond := #tempTimeMilliseconds MOD #MS_PER_SECOND;

     // check if value is greater then zero and add to result string without leading "+"
     IF (#tempMillisecond > #NO_REMAINDER) THEN
       #stringMilliSecond := DELETE(IN := DINT_TO_STRING(#tempMillisecond), L := #NUMBER_OF_CHAR_TO_DEL, P := #FIRST_POSITION);
       #tempTimeResult := CONCAT(IN1 := #stringMilliSecond, IN2 := 'MS');
     END_IF;

     // check if value is greater then zero and add to result string without leading "+"
     IF (#tempSecond > #NO_REMAINDER) THEN
       #stringSecond := DELETE(IN := DINT_TO_STRING(#tempSecond), L := #NUMBER_OF_CHAR_TO_DEL, P := #FIRST_POSITION);
       #tempTimeResult := CONCAT(IN1 := #stringSecond, IN2 := 'S', IN3 := #tempTimeResult);
     END_IF;

     // check if value is greater then zero and add to result string without leading "+"
     IF (#tempMinutes > #NO_REMAINDER) THEN
       #stringMinute := DELETE(IN := DINT_TO_STRING(#tempMinutes), L := #NUMBER_OF_CHAR_TO_DEL, P := #FIRST_POSITION);
       #tempTimeResult := CONCAT(IN1 := #stringMinute, IN2 := 'M', IN3 := #tempTimeResult);
     END_IF;

     // check if value is greater then zero and add to result string without leading "+"
     IF (#tempHours > #NO_REMAINDER) THEN
       #stringHour := DELETE(IN := DINT_TO_STRING(#tempHours), L := #NUMBER_OF_CHAR_TO_DEL, P := #FIRST_POSITION);
       #tempTimeResult := CONCAT(IN1 := #stringHour, IN2 := 'H', IN3 := #tempTimeResult);
     END_IF;

     // check if value is greater then zero and add to result string without leading "+"
     IF (#tempDays > #NO_REMAINDER) THEN
       #stringDay := DELETE(IN := DINT_TO_STRING(#tempDays), L := #NUMBER_OF_CHAR_TO_DEL, P := #FIRST_POSITION);
       #tempTimeResult := CONCAT(IN1 := #stringDay, IN2 := 'D', IN3 := #tempTimeResult);
     END_IF;
   END_REGION

   REGION OUTPUTS
     #LGF_TimeToString := #tempTimeResult;
     //ENO mechanism is not used - forced to true.
     ENO := TRUE;
   END_REGION
END_FUNCTION

FUNCTION "LGF_DTLToString_ISO" : String   // FC10083, SCL
TITLE = LGF_DTLtoString_ISO
{ S7_Optimized_Access := 'TRUE' }
AUTHOR : Siemens_Digital_Industry
FAMILY : LGF
NAME : LGF_DTLtoString_ISO
// This function converts a date of data type DTL into a character string of data type STRING in international format (YYYY MM DD…).
   VAR_INPUT
      "date" : DTL;   // Date to convert as DTL tag
      separator : Char;   // Separator between the components of the output date.
   END_VAR
   VAR_TEMP
      tempString : String;   // Temp string to setup the date string
      tempIndex : DInt;   // Temp iterator for replacing withspaces with '0' in nanosecondstring
   END_VAR
   // Ret_Val : Output string in accordance with the ISO 8601 format. Example: `2019-01-22 14:06:51.524621000`.
   VAR CONSTANT
      CONVERT_SIZE_YEAR : USInt := 4;   // Number of character positions for Year
      CONVERT_SIZE_MONTH_DAY_HOUR_MINUTE_SECOND : USInt := 2;   // Number of character positions for Month, Day, Minute and Second
      CONVERT_SIZE_NANOSECOND : USInt := 9;   // Number of character positions for Nanoseconds
      CONVERT_PRECISION : USInt := 0;   // Number of decimal places to convert
      CONVERT_FORMAT_TO_STRING : Word := 16#0000;   // Output format of the characters
      CONVERT_START_POSITION_YEAR : UInt := 1;   // Character starting in string at which position the result is written.
      CONVERT_START_POSITION_MONTH : UInt := 6;   // Character starting in string at which position the result is written.
      CONVERT_START_POSITION_DAY : UInt := 9;   // Character starting in string at which position the result is written.
      CONVERT_START_POSITION_HOUR : UInt := 12;   // Character starting in string at which position the result is written.
      CONVERT_START_POSITION_MINUTE : UInt := 15;   // Character starting in string at which position the result is written.
      CONVERT_START_POSITION_SECOND : UInt := 18;   // Character starting in string at which position the result is written.
      CONVERT_START_POSITION_NANOSECOND : UInt := 21;   // Character starting in string at which position the result is written.
      SEPARATOR_POSITION_YEAR_MONTH : UInt := 5;   // Character starting in string at which position the result is written.
      SEPARATOR_POSITION_MONTH_DAY : UInt := 8;   // Character starting in string at which position the result is written.
      SEPARATOR_POSITION_HOUR_MINUTE : UInt := 14;   // Character starting in string at which position the result is written.
      SEPARATOR_POSITION_MINUTE_SECOND : UInt := 17;   // Character starting in string at which position the result is written.
      SEPARATOR_POSITION_SECOND_NANOSECOND : UInt := 20;   // Character starting in string at which position the result is written.
      SEPARATOR_NANOSECOND : Char := '.';   // Seperator for Nanosecond
      SEPARATOR_TIME : Char := ':';   // Seperator for Time
      SEPARATOR_DATE : Char := '-';   // Default separator for Date
      REPLACE_NANOSECOND_COUNT : DInt := 8;   // Number of Nonosecond characters to be checked for replacing withspaces wit '0'
   END_VAR
BEGIN
   REGION BLOCK INFO HEADER
     //===============================================================================
     // SIEMENS AG / (c)Copyright 2019
     //-------------------------------------------------------------------------------
     // Title:            LGF_DTLtoString_ISO
     // Comment/Function: This function converts a date of data type DTL into a character string of data type STRING in international format (YYYY MM DD…).
     // Library/Family:   LGF (Library General Functions)
     // Author:           Siemens Digital Industry Support
     // Tested with:      S7-PLCSIM Advanced V2.0 SP1
     // Engineering:      TIA Portal V15.1
     // Restrictions:     ENO mechanism is not used, no error handling
     // Requirements:     PLC (S7-1200 / S7-1500)
     //-------------------------------------------------------------------------------
     // Change log table:
     // Version  | Date       | Expert in charge       | Changes applied
     //----------|------------|------------------------|------------------------------
     // 01.00.00 | 15.06.2016 | Siemens Industry Online Support
     //                         First released version
     // 01.00.01 | 02.01.2017 | Siemens Industry Online Support
     //                         Upgrade: TIA Portal V14 Update 1
     // 01.00.02 | 17.08.2018 | Siemens Industry Online Support
     //                         Upgrade: TIA V15 Update 2
     // 01.00.03 | 23.11.2018 | Siemens Industry Online Support
     //                         Upgrade: TIA V15.1
     // 01.00.04 | 17.07.2019 | Simatic Systems Support
     //                         Bugfix - nanosecond precision and '0' filling
     // 01.00.05 | 18.07.2019 | Simatic Systems Support
     //                         Renamed from "LGF_DTLtoString" to "LGF_DTLtoString_ISO"
     //                         Split into two blocks, removed "format" input
     // 03.00.00 | 23.04.2020 | Simatic Systems Support | Set version to V3.0.0
     //                         Harmonize the version of the whole library
     // 03.00.01 | 23.02.2021 | Simatic Systems Support
     //                         Insert documentation
     //=============================================================================
   END_REGION Block info header

   REGION DESCRIPTION
     (/*The block reads a date of data type DTL and converts the individual components of the date (year, month, day, hour…) into a character string and outputs it in international format. The separator between the components of the date is variable.

   ##### International format (ISO 8601):

   {.imagePageWidth}
   ![LGF_DTLtoString_ISO - Structure of the character string in accordance with ISO 8601](LGF_DTLtoString_ISO.png "LGF_DTLtoString_ISO - Structure of the character string in accordance with ISO 8601")

   ##### Separator:

   At the input parameter `separatorDate`, you specify the separator between the components of the calendar date.

   ##### Example:

   * separatorDate = `/` - outString = `2016/03/16…`
   * separatorDate = `-` - outString = `2016-03-16…`*/)
   END_REGION DESCRIPTION

   REGION INITIALISATION
     #tempString := '';
   END_REGION

   REGION CONVERTER
     // Set format parameters for output string
     // International ISO 8601
     // DTL  | Y| Y| Y| Y| -| M| M| -| D| D|  | H| H| :| M| M| :| S| S| .|NS|NS|NS|NS|NS|NS|NS|NS|NS
     // -----|--|--|--|--|--|--|--|--|--|--|--|--|--|--|--|--|--|--|--|--|--|--|--|--|--|--|--|--|--
     // Pos  | 1| 2| 3| 4| 5| 6| 7| 8| 9|10|11|12|13|14|15|16|17|18|19|20|21|22|23|24|25|26|27|28|29

     // Convert "Value" into "String" and place at the right position
     VAL_STRG(FORMAT := #CONVERT_FORMAT_TO_STRING,
              IN     := #date.YEAR,
              P      := #CONVERT_START_POSITION_YEAR,
              PREC   := #CONVERT_PRECISION,
              SIZE   := #CONVERT_SIZE_YEAR,
              OUT    => #tempString);    // DTL YEAR --> String --> #tempPosYear

     VAL_STRG(FORMAT := #CONVERT_FORMAT_TO_STRING,
              IN     := #date.MONTH,
              P      := #CONVERT_START_POSITION_MONTH,
              PREC   := #CONVERT_PRECISION,
              SIZE   := #CONVERT_SIZE_MONTH_DAY_HOUR_MINUTE_SECOND,
              OUT    => #tempString);     // DTL MONTH --> String --> #tempPosMonth

     VAL_STRG(FORMAT := #CONVERT_FORMAT_TO_STRING,
              IN     := #date.DAY,
              P      := #CONVERT_START_POSITION_DAY,
              PREC   := #CONVERT_PRECISION,
              SIZE   := #CONVERT_SIZE_MONTH_DAY_HOUR_MINUTE_SECOND,
              OUT    => #tempString);     // DTL DAY --> String --> #tempPosDay

     VAL_STRG(FORMAT := #CONVERT_FORMAT_TO_STRING,
              IN     := #date.HOUR,
              P      := #CONVERT_START_POSITION_HOUR,
              PREC   := #CONVERT_PRECISION,
              SIZE   := #CONVERT_SIZE_MONTH_DAY_HOUR_MINUTE_SECOND,
              OUT    => #tempString);     // DTL HOUR --> String --> #tempPosHour

     VAL_STRG(FORMAT := #CONVERT_FORMAT_TO_STRING,
              IN     := #date.MINUTE,
              P      := #CONVERT_START_POSITION_MINUTE,
              PREC   := #CONVERT_PRECISION,
              SIZE   := #CONVERT_SIZE_MONTH_DAY_HOUR_MINUTE_SECOND,
              OUT    => #tempString);     // DTL MINUTE --> String --> #tempPosMinute

     VAL_STRG(FORMAT := #CONVERT_FORMAT_TO_STRING,
              IN     := #date.SECOND,
              P      := #CONVERT_START_POSITION_SECOND,
              PREC   := #CONVERT_PRECISION,
              SIZE   := #CONVERT_SIZE_MONTH_DAY_HOUR_MINUTE_SECOND,
              OUT    => #tempString);     // DTL SECOND --> String --> #tempPosSecond

     VAL_STRG(FORMAT := #CONVERT_FORMAT_TO_STRING,
              IN     := #date.NANOSECOND,
              P      := #CONVERT_START_POSITION_NANOSECOND,
              PREC   := #CONVERT_PRECISION,
              SIZE   := #CONVERT_SIZE_NANOSECOND,
              OUT    => #tempString);     // DTL NANOSECOND --> String --> #tempPosNanosecond

     // Place separators at the right position in the string
     IF #separator = '' THEN
       #tempString[#SEPARATOR_POSITION_YEAR_MONTH] := #SEPARATOR_DATE;
       #tempString[#SEPARATOR_POSITION_MONTH_DAY] := #SEPARATOR_DATE;
     ELSE
       #tempString[#SEPARATOR_POSITION_YEAR_MONTH] := #separator;
       #tempString[#SEPARATOR_POSITION_MONTH_DAY] := #separator;
     END_IF;
     #tempString[#SEPARATOR_POSITION_HOUR_MINUTE] := #SEPARATOR_TIME;
     #tempString[#SEPARATOR_POSITION_MINUTE_SECOND] := #SEPARATOR_TIME;
     #tempString[#SEPARATOR_POSITION_SECOND_NANOSECOND] := #SEPARATOR_NANOSECOND;

     // Correcting the string, due to the conversion of a leading "0" value into a "blank".
     // Replacing of "blank" by "0"
     IF (#tempString[#CONVERT_START_POSITION_MONTH] = ' ') THEN
       #tempString[#CONVERT_START_POSITION_MONTH] := '0';
     END_IF;

     IF (#tempString[#CONVERT_START_POSITION_DAY] = ' ') THEN
       #tempString[#CONVERT_START_POSITION_DAY] := '0';
     END_IF;

     IF (#tempString[#CONVERT_START_POSITION_HOUR] = ' ') THEN
       #tempString[#CONVERT_START_POSITION_HOUR] := '0';
     END_IF;

     IF (#tempString[#CONVERT_START_POSITION_MINUTE] = ' ') THEN
       #tempString[#CONVERT_START_POSITION_MINUTE] := '0';
     END_IF;

     IF (#tempString[#CONVERT_START_POSITION_SECOND] = ' ') THEN
       #tempString[#CONVERT_START_POSITION_SECOND] := '0';
     END_IF;

     FOR #tempIndex := 0 TO #REPLACE_NANOSECOND_COUNT DO
       IF (#tempString[UINT_TO_SINT(#CONVERT_START_POSITION_NANOSECOND) + #tempIndex] = ' ') THEN
         #tempString[UINT_TO_SINT(#CONVERT_START_POSITION_NANOSECOND) + #tempIndex] := '0';
       ELSE
         EXIT;
       END_IF;
     END_FOR;
   END_REGION

   REGION OUTPUTS
     #LGF_DTLToString_ISO := #tempString;
     // no error handling needed
     ENO := TRUE;
   END_REGION
END_FUNCTION

// folder: LMQTT

